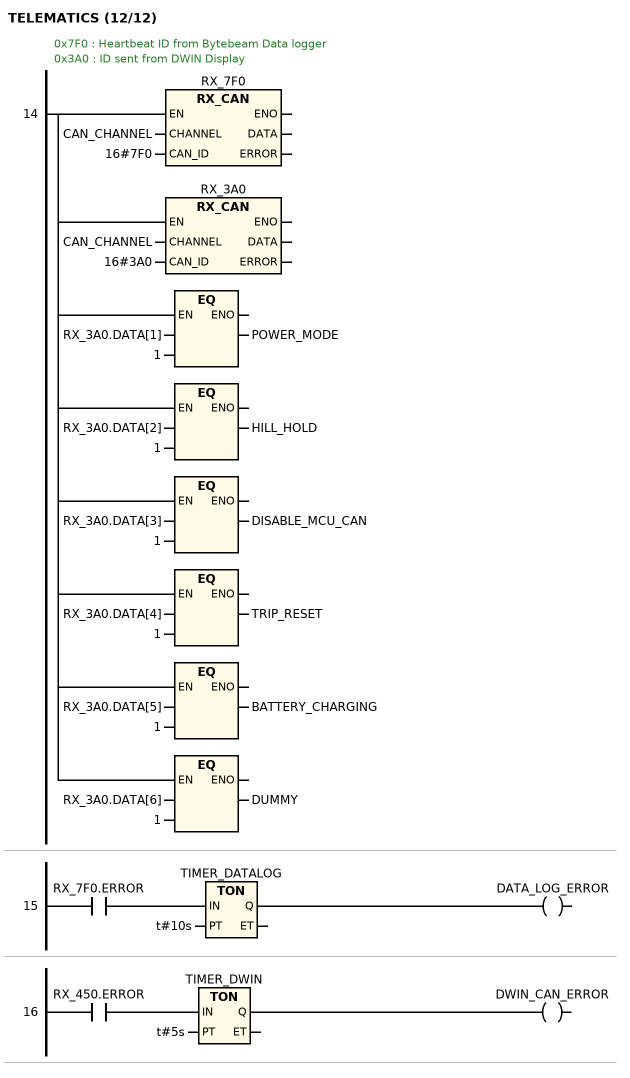
[picture p48: TELEMATICS (LD)]
_LD_ (* Ladder Diagram *)
NETWORK 1 (* CAN ID 301: Battery 1 data Message 1 *)
	*
		EN --- INT_TO_WORD(BATTERY1_POWER) => WB_BATTERY1_POWER.IN_WORD
		EN --- WB_BATTERY1_POWER:WORD_BYTE_CONVERSION(IN_WORD: WB_BATTERY1_POWER.IN_WORD)
		EN --- PACK(BATTERY1_CHARGING, BATTERY1_CAN_ERROR, 0, 0, 0, 0, 0, 0) => PACK_301.B4
		EN --- INT_TO_BYTE(BATTERY1_CAPACITY) => PACK_301.B5
		EN --- PACK_301:PACK_BYTES(B0: BATTERY1_SOC, B1: BATTERY1_SOH, B2: WB_BATTERY1_POWER.BYTE_H, B3: WB_BATTERY1_POWER.BYTE_L, B4: PACK_301.B4, B5: PACK_301.B5, B6: BATTERY1_NTC1, B7: BATTERY1_NTC2) => TX_301.DATA
NETWORK 2 (* CAN ID 303: Battery2 data *)
	*
		EN --- INT_TO_WORD(BATTERY2_POWER) => WB_BATTERY2_POWER.IN_WORD
		EN --- WB_BATTERY2_POWER:WORD_BYTE_CONVERSION(IN_WORD: WB_BATTERY2_POWER.IN_WORD)
		EN --- PACK(BATTERY2_CHARGING, BATTERY2_CAN_ERROR, 0, 0, 0, 0, 0, 0) => PACK_303.B4
		EN --- INT_TO_BYTE(BATTERY2_CAPACITY) => PACK_303.B5
		EN --- PACK_303:PACK_BYTES(B0: BATTERY2_SOC, B1: BATTERY2_SOH, B2: WB_BATTERY2_POWER.BYTE_H, B3: WB_BATTERY2_POWER.BYTE_L, B4: PACK_303.B4, B5: PACK_303.B5, B6: BATTERY2_NTC1, B7: BATTERY2_NTC2) => TX_303.DATA
NETWORK 3 (* CAN ID 305: ODO and TRIP Data *)
	*
		EN --- WB_HYDL_UPTIME:DWORD_BYTE_CONVERSION(INPUT_DWORD: HYDL_UP_TIME)
		EN --- WB_RUNTIME_MIN:DWORD_BYTE_CONVERSION(INPUT_DWORD: RUNTIME)
		EN --- PACK_305:PACK_BYTES(B0: WB_RUNTIME_MIN.BYTE_3, B1: WB_RUNTIME_MIN.BYTE_2, B2: WB_RUNTIME_MIN.BYTE_1, B3: WB_RUNTIME_MIN.BYTE_0, B4: WB_HYDL_UPTIME.BYTE_3, B5: WB_HYDL_UPTIME.BYTE_2, B6: WB_HYDL_UPTIME.BYTE_1, B7: WB_HYDL_UPTIME.BYTE_0) => TX_305.DATA
NETWORK 4 (* CAN ID 306: Basic Vehicle Data *)
	*
		EN --- WB_ODO_METERS:DWORD_BYTE_CONVERSION(INPUT_DWORD: ODO_METER)
		EN --- PACK_306:PACK_BYTES(B0: WB_ODO_METERS.BYTE_3, B1: WB_ODO_METERS.BYTE_2, B2: WB_ODO_METERS.BYTE_1, B3: WB_ODO_METERS.BYTE_0, B4: SPEED, B5: 0, B6: LOG_JX, B7: LOG_JY) => TX_306.DATA
NETWORK 5 (* CAN ID 307: Vehicle Specific parameter frame *)
	*
		EN --- PACK(MCU_IGNITION, NOT KILL_SWITCH, EM_SWITCH, HYDRAULIC_IGNITION, REVERSE, HIGH_SPEED, EM_BRAKE, POWER_MODE) => TX_307.DATA[0]
		EN --- PACK(JOY_ERROR, DATA_LOG_ERROR, DWIN_CAN_ERROR, 0, 0, 0, 0, 0) => TX_307.DATA[1]
		EN --- PACK(BATTERY1_IGNITION, BATTERY2_IGNITION, 0, BATTERY1_RELAY, BATTERY2_RELAY, IMU_ALERT, 0, 0) => TX_307.DATA[2]
		EN --- MOVE(X_ANGLE_BYTE) => TX_307.DATA[6]
		EN --- MOVE(Y_ANGLE_BYTE) => TX_307.DATA[7]
NETWORK 6 (* IMU DATA: 0x308 *)
	*
		EN --- PACK_308:PACK_BYTES(B0: Y_MAX_RETAIN, B1: Y_MIN_RETAIN, B2: X_MAX_RETAIN, B3: X_MIN_RETAIN, B4: Y_MAX_PEAK, B5: Y_MIN_PEAK, B6: X_MAX_PEAK, B7: X_MIN_PEAK) => TX_308.DATA
NETWORK 7 (* 409:- VEHICLE UP TIME (NOT SENDING TO BYTEBEAM) *)
	*
		EN --- WB_VEHICLE_UPTIME:DWORD_BYTE_CONVERSION(INPUT_DWORD: VEHICLE_UP_TIME)
		EN --- WB_VEHICLE_UPTIME_LT:DWORD_BYTE_CONVERSION(INPUT_DWORD: VEHICLE_UP_TIME_LT)
		EN --- PACK_409:PACK_BYTES(B0: WB_VEHICLE_UPTIME_LT.BYTE_3, B1: WB_VEHICLE_UPTIME_LT.BYTE_2, B2: WB_VEHICLE_UPTIME_LT.BYTE_1, B3: WB_VEHICLE_UPTIME_LT.BYTE_0, B4: WB_VEHICLE_UPTIME.BYTE_3, B5: WB_VEHICLE_UPTIME.BYTE_2, B6: WB_VEHICLE_UPTIME.BYTE_1, B7: WB_VEHICLE_UPTIME.BYTE_0) => TX_409.DATA
NETWORK 8 (* CAN ID 310: Motor 41 data Message 1 / CAN ID 311: Motor 41 data Message 2 *)
	*
		EN --- INT_TO_WORD(MOTOR_RPM[1]) => WB_RPM_1.IN_WORD
		EN --- WB_RPM_1:WORD_BYTE_CONVERSION(IN_WORD: WB_RPM_1.IN_WORD, BYTE_L => TX_310.DATA[1]) => TX_310.DATA[0]
		EN --- INT_TO_WORD(MOTOR_POWER[1]) => WB_POWER_1.IN_WORD
		EN --- WB_POWER_1:WORD_BYTE_CONVERSION(IN_WORD: WB_POWER_1.IN_WORD, BYTE_L => TX_310.DATA[3]) => TX_310.DATA[2]
		EN --- WB_PHASE_1:WORD_BYTE_CONVERSION(IN_WORD: MOTOR_PHASE_CURRENT[1], BYTE_L => TX_310.DATA[5]) => TX_310.DATA[4]
		EN --- MOVE(MOTOR_TEMPERATURE[1]) => TX_310.DATA[6]
		EN --- MOVE(MCU_TEMPERATURE[1]) => TX_310.DATA[7]
		EN --- INT_TO_WORD(MOTOR_TARGET_RPM[1]) => WB_TARGET_RPM_1.IN_WORD
		EN --- WB_TARGET_RPM_1:WORD_BYTE_CONVERSION(IN_WORD: WB_TARGET_RPM_1.IN_WORD)
		EN --- WORD_TO_BYTE(MOTOR_OBD_ARRAY[1]) => OBD1_BYTE
		EN --- PACK(MCU_CAN_ERROR[1], 0, 0, 0, 0, 0, 0, 0) => PACK_311.B2
		EN --- PACK_311:PACK_BYTES(B0: WB_TARGET_RPM_1.BYTE_H, B1: WB_TARGET_RPM_1.BYTE_L, B2: PACK_311.B2, B3: OBD1_BYTE, B4: MOTOR1_FAULT_ARRAY[1], B5: MOTOR1_FAULT_ARRAY[2], B6: MOTOR1_FAULT_ARRAY[3], B7: MOTOR1_FAULT_ARRAY[4]) => TX_311.DATA
NETWORK 9 (* CAN ID 312: Motor 42 data Message 1 / CAN ID 313: Motor 42 data Message 2 *)
	*
		EN --- INT_TO_WORD(MOTOR_RPM[2]) => WB_RPM_2.IN_WORD
		EN --- WB_RPM_2:WORD_BYTE_CONVERSION(IN_WORD: WB_RPM_2.IN_WORD, BYTE_L => TX_312.DATA[1]) => TX_312.DATA[0]
		EN --- INT_TO_WORD(MOTOR_POWER[2]) => WB_POWER_2.IN_WORD
		EN --- WB_POWER_2:WORD_BYTE_CONVERSION(IN_WORD: WB_POWER_2.IN_WORD, BYTE_L => TX_312.DATA[3]) => TX_312.DATA[2]
		EN --- WB_PHASE_2:WORD_BYTE_CONVERSION(IN_WORD: MOTOR_PHASE_CURRENT[2], BYTE_L => TX_312.DATA[5]) => TX_312.DATA[4]
		EN --- MOVE(MOTOR_TEMPERATURE[2]) => TX_312.DATA[6]
		EN --- MOVE(MCU_TEMPERATURE[2]) => TX_312.DATA[7]
		EN --- INT_TO_WORD(MOTOR_TARGET_RPM[2]) => WB_TARGET_RPM_2.IN_WORD
		EN --- WB_TARGET_RPM_2:WORD_BYTE_CONVERSION(IN_WORD: WB_TARGET_RPM_2.IN_WORD)
		EN --- WB_OBD_2:WORD_BYTE_CONVERSION(IN_WORD: MOTOR_OBD_ARRAY[2])
		EN --- WORD_TO_BYTE(MOTOR_OBD_ARRAY[2]) => OBD2_BYTE
		EN --- PACK(MCU_CAN_ERROR[2], 0, 0, 0, 0, 0, 0, 0) => TX_313.DATA[2]
		EN --- PACK_313:PACK_BYTES(B0: WB_TARGET_RPM_2.BYTE_H, B1: WB_TARGET_RPM_2.BYTE_L, B2: TX_313.DATA[2], B3: OBD2_BYTE, B4: MOTOR2_FAULT_ARRAY[1], B5: MOTOR2_FAULT_ARRAY[2], B6: MOTOR2_FAULT_ARRAY[3], B7: MOTOR2_FAULT_ARRAY[4]) => TX_313.DATA
NETWORK 10 (* CAN ID 31A: Motor 46 data Message 1 / CAN ID 31B: Motor 46 data Message 2 *)
	*
		EN --- INT_TO_WORD(MOTOR_RPM[6]) => WB_RPM_6.IN_WORD
		EN --- WB_RPM_6:WORD_BYTE_CONVERSION(IN_WORD: WB_RPM_6.IN_WORD, BYTE_L => TX_31A.DATA[1]) => TX_31A.DATA[0]
		EN --- INT_TO_WORD(MOTOR_POWER[6]) => WB_POWER_6.IN_WORD
		EN --- WB_POWER_6:WORD_BYTE_CONVERSION(IN_WORD: WB_POWER_6.IN_WORD, BYTE_L => TX_31A.DATA[3]) => TX_31A.DATA[2]
		EN --- WB_PHASE_6:WORD_BYTE_CONVERSION(IN_WORD: MOTOR_PHASE_CURRENT[6], BYTE_L => TX_31A.DATA[5]) => TX_31A.DATA[4]
		EN --- MOVE(MOTOR_TEMPERATURE[6]) => TX_31A.DATA[6]
		EN --- MOVE(MCU_TEMPERATURE[6]) => TX_31A.DATA[7]
		EN --- INT_TO_WORD(MOTOR_TARGET_RPM[6]) => WB_TARGET_RPM_6.IN_WORD
		EN --- WB_TARGET_RPM_6:WORD_BYTE_CONVERSION(IN_WORD: WB_TARGET_RPM_6.IN_WORD)
		EN --- WB_OBD_6:WORD_BYTE_CONVERSION(IN_WORD: MOTOR_OBD_ARRAY[6])
		EN --- WORD_TO_BYTE(MOTOR_OBD_ARRAY[6]) => OBD6_BYTE
		EN --- PACK(MCU_CAN_ERROR[6], 0, 0, 0, 0, 0, 0, 0) => TX_31B.DATA[2]
		EN --- PACK_31B:PACK_BYTES(B0: WB_TARGET_RPM_6.BYTE_H, B1: WB_TARGET_RPM_6.BYTE_L, B2: TX_31B.DATA[2], B3: OBD6_BYTE, B4: MOTOR6_FAULT_ARRAY[1], B5: MOTOR6_FAULT_ARRAY[2], B6: MOTOR6_FAULT_ARRAY[3], B7: MOTOR6_FAULT_ARRAY[4]) => TX_31B.DATA
NETWORK 11 (* CAN ID 262: BATTERY CHARGING TIME *)
	*
		EN --- REAL_TO_WORD(BATTERY1_FULLCHARGE_MIN) => WD_BATTERY1_FULLCHARGE_MIN
		EN --- REAL_TO_WORD(BATTERY2_FULLCHARGE_MIN) => WD_BATTERY2_FULLCHARGE_MIN
		EN --- WB_FULLCHARGE1_MIN:WORD_BYTE_CONVERSION(IN_WORD: WD_BATTERY1_FULLCHARGE_MIN)
		EN --- WB_FULLCHARGE2_MIN:WORD_BYTE_CONVERSION(IN_WORD: WD_BATTERY2_FULLCHARGE_MIN)
		EN --- PACK_262:PACK_BYTES(B0: WB_FULLCHARGE1_MIN.BYTE_H, B1: WB_FULLCHARGE1_MIN.BYTE_L, B2: WB_FULLCHARGE2_MIN.BYTE_H, B3: WB_FULLCHARGE2_MIN.BYTE_L, B4: 0, B5: 0, B6: 0, B7: 0) => TX_262.DATA
NETWORK 12 (* TO BYTEBEAM *)
	[/TIMER_TX_1.Q] - TIMER_TX_1:TON(IN: *, PT: t#490ms)
		EN --- TX_300:CAN_TX(ENABLE: TRUE, CHANNEL: CAN_CHANNEL, ID: 16#300, DATA: META_FRAME)
		EN --- TX_301:CAN_TX(ENABLE: TRUE, CHANNEL: CAN_CHANNEL, ID: 16#301, DATA: TX_301.DATA)
		EN --- TX_303:CAN_TX(ENABLE: TRUE, CHANNEL: CAN_CHANNEL, ID: 16#303, DATA: TX_303.DATA)
		EN --- TX_306:CAN_TX(ENABLE: TRUE, CHANNEL: CAN_CHANNEL, ID: 16#306, DATA: TX_306.DATA)
		EN --- TX_307:CAN_TX(ENABLE: TRUE, CHANNEL: CAN_CHANNEL, ID: 16#307, DATA: TX_307.DATA)
		EN --- TX_310:CAN_TX(ENABLE: TRUE, CHANNEL: CAN_CHANNEL, ID: 16#310, DATA: TX_310.DATA)
		EN --- TX_311:CAN_TX(ENABLE: TRUE, CHANNEL: CAN_CHANNEL, ID: 16#311, DATA: TX_311.DATA)
		EN --- TX_312:CAN_TX(ENABLE: TRUE, CHANNEL: CAN_CHANNEL, ID: 16#312, DATA: TX_312.DATA)
		EN --- TX_313:CAN_TX(ENABLE: TRUE, CHANNEL: CAN_CHANNEL, ID: 16#313, DATA: TX_313.DATA)
		EN --- TX_31A:CAN_TX(ENABLE: TRUE, CHANNEL: CAN_CHANNEL, ID: 16#31A, DATA: TX_31A.DATA)
		EN --- TX_31B:CAN_TX(ENABLE: TRUE, CHANNEL: CAN_CHANNEL, ID: 16#31B, DATA: TX_31B.DATA)
		EN --- TX_308:CAN_TX(ENABLE: TRUE, CHANNEL: CAN_CHANNEL, ID: 16#308, DATA: TX_308.DATA)
		EN --- TX_305:CAN_TX(ENABLE: TRUE, CHANNEL: CAN_CHANNEL, ID: 16#305, DATA: TX_305.DATA)
NETWORK 13 (* TO DISPLAY *)
	[/TIMER_TX_2.Q] - TIMER_TX_2:TON(IN: *, PT: t#50ms)
		EN --- TX_400:CAN_TX(ENABLE: TRUE, CHANNEL: CAN_CHANNEL, ID: 16#400, DATA: META_FRAME)
		EN --- TX_401:CAN_TX(ENABLE: TRUE, CHANNEL: CAN_CHANNEL, ID: 16#401, DATA: TX_301.DATA)
		EN --- TX_403:CAN_TX(ENABLE: TRUE, CHANNEL: CAN_CHANNEL, ID: 16#403, DATA: TX_303.DATA)
		EN --- TX_406:CAN_TX(ENABLE: TRUE, CHANNEL: CAN_CHANNEL, ID: 16#406, DATA: TX_306.DATA)
		EN --- TX_407:CAN_TX(ENABLE: TRUE, CHANNEL: CAN_CHANNEL, ID: 16#407, DATA: TX_307.DATA)
		EN --- TX_410:CAN_TX(ENABLE: TRUE, CHANNEL: CAN_CHANNEL, ID: 16#410, DATA: TX_310.DATA)
		EN --- TX_411:CAN_TX(ENABLE: TRUE, CHANNEL: CAN_CHANNEL, ID: 16#411, DATA: TX_311.DATA)
		EN --- TX_412:CAN_TX(ENABLE: TRUE, CHANNEL: CAN_CHANNEL, ID: 16#412, DATA: TX_312.DATA)
		EN --- TX_413:CAN_TX(ENABLE: TRUE, CHANNEL: CAN_CHANNEL, ID: 16#413, DATA: TX_313.DATA)
		EN --- TX_41A:CAN_TX(ENABLE: TRUE, CHANNEL: CAN_CHANNEL, ID: 16#41A, DATA: TX_31A.DATA)
		EN --- TX_41B:CAN_TX(ENABLE: TRUE, CHANNEL: CAN_CHANNEL, ID: 16#41B, DATA: TX_31B.DATA)
		EN --- TX_262:CAN_TX(ENABLE: TRUE, CHANNEL: CAN_CHANNEL, ID: 16#262, DATA: TX_262.DATA)
		EN --- TX_408:CAN_TX(ENABLE: TRUE, CHANNEL: CAN_CHANNEL, ID: 16#408, DATA: TX_308.DATA)
		EN --- TX_405:CAN_TX(ENABLE: TRUE, CHANNEL: CAN_CHANNEL, ID: 16#405, DATA: TX_305.DATA)
		EN --- TX_409:CAN_TX(ENABLE: TRUE, CHANNEL: CAN_CHANNEL, ID: 16#409, DATA: TX_409.DATA)
NETWORK 14 (* 0x7F0 : Heartbeat ID from Bytebeam Data logger / 0x3A0 : ID sent from DWIN Display *)
	*
		EN --- RX_7F0:RX_CAN(CHANNEL: CAN_CHANNEL, CAN_ID: 16#7F0)
		EN --- RX_3A0:RX_CAN(CHANNEL: CAN_CHANNEL, CAN_ID: 16#3A0)
		EN --- EQ(RX_3A0.DATA[1], 1) => POWER_MODE
		EN --- EQ(RX_3A0.DATA[2], 1) => HILL_HOLD
		EN --- EQ(RX_3A0.DATA[3], 1) => DISABLE_MCU_CAN
		EN --- EQ(RX_3A0.DATA[4], 1) => TRIP_RESET
		EN --- EQ(RX_3A0.DATA[5], 1) => BATTERY_CHARGING
		EN --- EQ(RX_3A0.DATA[6], 1) => DUMMY
NETWORK 15
	[RX_7F0.ERROR] - TIMER_DATALOG:TON(IN: *, PT: t#10s) --- (DATA_LOG_ERROR)
NETWORK 16
	[RX_450.ERROR] - TIMER_DWIN:TON(IN: *, PT: t#5s) --- (DWIN_CAN_ERROR)
_END_LD_
(* the same logic as Structured Text *)
(* Network 1: CAN ID 301: Battery 1 data Message 1 *)
WB_BATTERY1_POWER.IN_WORD := INT_TO_WORD(BATTERY1_POWER);
WB_BATTERY1_POWER(IN_WORD := WB_BATTERY1_POWER.IN_WORD);
PACK_301.B4 := PACK(BATTERY1_CHARGING, BATTERY1_CAN_ERROR, 0, 0, 0, 0, 0, 0);
PACK_301.B5 := INT_TO_BYTE(BATTERY1_CAPACITY);
PACK_301(B0 := BATTERY1_SOC, B1 := BATTERY1_SOH, B2 := WB_BATTERY1_POWER.BYTE_H, B3 := WB_BATTERY1_POWER.BYTE_L, B4 := PACK_301.B4, B5 := PACK_301.B5, B6 := BATTERY1_NTC1, B7 := BATTERY1_NTC2);
TX_301.DATA := PACK_301.CAN_DATA;
(* Network 2: CAN ID 303: Battery2 data *)
WB_BATTERY2_POWER.IN_WORD := INT_TO_WORD(BATTERY2_POWER);
WB_BATTERY2_POWER(IN_WORD := WB_BATTERY2_POWER.IN_WORD);
PACK_303.B4 := PACK(BATTERY2_CHARGING, BATTERY2_CAN_ERROR, 0, 0, 0, 0, 0, 0);
PACK_303.B5 := INT_TO_BYTE(BATTERY2_CAPACITY);
PACK_303(B0 := BATTERY2_SOC, B1 := BATTERY2_SOH, B2 := WB_BATTERY2_POWER.BYTE_H, B3 := WB_BATTERY2_POWER.BYTE_L, B4 := PACK_303.B4, B5 := PACK_303.B5, B6 := BATTERY2_NTC1, B7 := BATTERY2_NTC2);
TX_303.DATA := PACK_303.CAN_DATA;
(* Network 3: CAN ID 305: ODO and TRIP Data *)
WB_HYDL_UPTIME(INPUT_DWORD := HYDL_UP_TIME);
WB_RUNTIME_MIN(INPUT_DWORD := RUNTIME);
PACK_305(B0 := WB_RUNTIME_MIN.BYTE_3, B1 := WB_RUNTIME_MIN.BYTE_2, B2 := WB_RUNTIME_MIN.BYTE_1, B3 := WB_RUNTIME_MIN.BYTE_0, B4 := WB_HYDL_UPTIME.BYTE_3, B5 := WB_HYDL_UPTIME.BYTE_2, B6 := WB_HYDL_UPTIME.BYTE_1, B7 := WB_HYDL_UPTIME.BYTE_0);
TX_305.DATA := PACK_305.CAN_DATA;
(* Network 4: CAN ID 306: Basic Vehicle Data *)
WB_ODO_METERS(INPUT_DWORD := ODO_METER);
PACK_306(B0 := WB_ODO_METERS.BYTE_3, B1 := WB_ODO_METERS.BYTE_2, B2 := WB_ODO_METERS.BYTE_1, B3 := WB_ODO_METERS.BYTE_0, B4 := SPEED, B5 := 0, B6 := LOG_JX, B7 := LOG_JY);
TX_306.DATA := PACK_306.CAN_DATA;
(* Network 5: CAN ID 307: Vehicle Specific parameter frame *)
TX_307.DATA[0] := PACK(MCU_IGNITION, NOT KILL_SWITCH, EM_SWITCH, HYDRAULIC_IGNITION, REVERSE, HIGH_SPEED, EM_BRAKE, POWER_MODE);
TX_307.DATA[1] := PACK(JOY_ERROR, DATA_LOG_ERROR, DWIN_CAN_ERROR, 0, 0, 0, 0, 0);
TX_307.DATA[2] := PACK(BATTERY1_IGNITION, BATTERY2_IGNITION, 0, BATTERY1_RELAY, BATTERY2_RELAY, IMU_ALERT, 0, 0);
TX_307.DATA[6] := X_ANGLE_BYTE;
TX_307.DATA[7] := Y_ANGLE_BYTE;
(* Network 6: IMU DATA: 0x308 *)
PACK_308(B0 := Y_MAX_RETAIN, B1 := Y_MIN_RETAIN, B2 := X_MAX_RETAIN, B3 := X_MIN_RETAIN, B4 := Y_MAX_PEAK, B5 := Y_MIN_PEAK, B6 := X_MAX_PEAK, B7 := X_MIN_PEAK);
TX_308.DATA := PACK_308.CAN_DATA;
(* Network 7: 409:- VEHICLE UP TIME (NOT SENDING TO BYTEBEAM) *)
WB_VEHICLE_UPTIME(INPUT_DWORD := VEHICLE_UP_TIME);
WB_VEHICLE_UPTIME_LT(INPUT_DWORD := VEHICLE_UP_TIME_LT);
PACK_409(B0 := WB_VEHICLE_UPTIME_LT.BYTE_3, B1 := WB_VEHICLE_UPTIME_LT.BYTE_2, B2 := WB_VEHICLE_UPTIME_LT.BYTE_1, B3 := WB_VEHICLE_UPTIME_LT.BYTE_0, B4 := WB_VEHICLE_UPTIME.BYTE_3, B5 := WB_VEHICLE_UPTIME.BYTE_2, B6 := WB_VEHICLE_UPTIME.BYTE_1, B7 := WB_VEHICLE_UPTIME.BYTE_0);
TX_409.DATA := PACK_409.CAN_DATA;
(* Network 8: CAN ID 310: Motor 41 data Message 1 / CAN ID 311: Motor 41 data Message 2 *)
WB_RPM_1.IN_WORD := INT_TO_WORD(MOTOR_RPM[1]);
WB_RPM_1(IN_WORD := WB_RPM_1.IN_WORD);
TX_310.DATA[1] := WB_RPM_1.BYTE_L;
TX_310.DATA[0] := WB_RPM_1.BYTE_H;
WB_POWER_1.IN_WORD := INT_TO_WORD(MOTOR_POWER[1]);
WB_POWER_1(IN_WORD := WB_POWER_1.IN_WORD);
TX_310.DATA[3] := WB_POWER_1.BYTE_L;
TX_310.DATA[2] := WB_POWER_1.BYTE_H;
WB_PHASE_1(IN_WORD := MOTOR_PHASE_CURRENT[1]);
TX_310.DATA[5] := WB_PHASE_1.BYTE_L;
TX_310.DATA[4] := WB_PHASE_1.BYTE_H;
TX_310.DATA[6] := MOTOR_TEMPERATURE[1];
TX_310.DATA[7] := MCU_TEMPERATURE[1];
WB_TARGET_RPM_1.IN_WORD := INT_TO_WORD(MOTOR_TARGET_RPM[1]);
WB_TARGET_RPM_1(IN_WORD := WB_TARGET_RPM_1.IN_WORD);
OBD1_BYTE := WORD_TO_BYTE(MOTOR_OBD_ARRAY[1]);
PACK_311.B2 := PACK(MCU_CAN_ERROR[1], 0, 0, 0, 0, 0, 0, 0);
PACK_311(B0 := WB_TARGET_RPM_1.BYTE_H, B1 := WB_TARGET_RPM_1.BYTE_L, B2 := PACK_311.B2, B3 := OBD1_BYTE, B4 := MOTOR1_FAULT_ARRAY[1], B5 := MOTOR1_FAULT_ARRAY[2], B6 := MOTOR1_FAULT_ARRAY[3], B7 := MOTOR1_FAULT_ARRAY[4]);
TX_311.DATA := PACK_311.CAN_DATA;
(* Network 9: CAN ID 312: Motor 42 data Message 1 / CAN ID 313: Motor 42 data Message 2 *)
WB_RPM_2.IN_WORD := INT_TO_WORD(MOTOR_RPM[2]);
WB_RPM_2(IN_WORD := WB_RPM_2.IN_WORD);
TX_312.DATA[1] := WB_RPM_2.BYTE_L;
TX_312.DATA[0] := WB_RPM_2.BYTE_H;
WB_POWER_2.IN_WORD := INT_TO_WORD(MOTOR_POWER[2]);
WB_POWER_2(IN_WORD := WB_POWER_2.IN_WORD);
TX_312.DATA[3] := WB_POWER_2.BYTE_L;
TX_312.DATA[2] := WB_POWER_2.BYTE_H;
WB_PHASE_2(IN_WORD := MOTOR_PHASE_CURRENT[2]);
TX_312.DATA[5] := WB_PHASE_2.BYTE_L;
TX_312.DATA[4] := WB_PHASE_2.BYTE_H;
TX_312.DATA[6] := MOTOR_TEMPERATURE[2];
TX_312.DATA[7] := MCU_TEMPERATURE[2];
WB_TARGET_RPM_2.IN_WORD := INT_TO_WORD(MOTOR_TARGET_RPM[2]);
WB_TARGET_RPM_2(IN_WORD := WB_TARGET_RPM_2.IN_WORD);
WB_OBD_2(IN_WORD := MOTOR_OBD_ARRAY[2]);
OBD2_BYTE := WORD_TO_BYTE(MOTOR_OBD_ARRAY[2]);
TX_313.DATA[2] := PACK(MCU_CAN_ERROR[2], 0, 0, 0, 0, 0, 0, 0);
PACK_313(B0 := WB_TARGET_RPM_2.BYTE_H, B1 := WB_TARGET_RPM_2.BYTE_L, B2 := TX_313.DATA[2], B3 := OBD2_BYTE, B4 := MOTOR2_FAULT_ARRAY[1], B5 := MOTOR2_FAULT_ARRAY[2], B6 := MOTOR2_FAULT_ARRAY[3], B7 := MOTOR2_FAULT_ARRAY[4]);
TX_313.DATA := PACK_313.CAN_DATA;
(* Network 10: CAN ID 31A: Motor 46 data Message 1 / CAN ID 31B: Motor 46 data Message 2 *)
WB_RPM_6.IN_WORD := INT_TO_WORD(MOTOR_RPM[6]);
WB_RPM_6(IN_WORD := WB_RPM_6.IN_WORD);
TX_31A.DATA[1] := WB_RPM_6.BYTE_L;
TX_31A.DATA[0] := WB_RPM_6.BYTE_H;
WB_POWER_6.IN_WORD := INT_TO_WORD(MOTOR_POWER[6]);
WB_POWER_6(IN_WORD := WB_POWER_6.IN_WORD);
TX_31A.DATA[3] := WB_POWER_6.BYTE_L;
TX_31A.DATA[2] := WB_POWER_6.BYTE_H;
WB_PHASE_6(IN_WORD := MOTOR_PHASE_CURRENT[6]);
TX_31A.DATA[5] := WB_PHASE_6.BYTE_L;
TX_31A.DATA[4] := WB_PHASE_6.BYTE_H;
TX_31A.DATA[6] := MOTOR_TEMPERATURE[6];
TX_31A.DATA[7] := MCU_TEMPERATURE[6];
WB_TARGET_RPM_6.IN_WORD := INT_TO_WORD(MOTOR_TARGET_RPM[6]);
WB_TARGET_RPM_6(IN_WORD := WB_TARGET_RPM_6.IN_WORD);
WB_OBD_6(IN_WORD := MOTOR_OBD_ARRAY[6]);
OBD6_BYTE := WORD_TO_BYTE(MOTOR_OBD_ARRAY[6]);
TX_31B.DATA[2] := PACK(MCU_CAN_ERROR[6], 0, 0, 0, 0, 0, 0, 0);
PACK_31B(B0 := WB_TARGET_RPM_6.BYTE_H, B1 := WB_TARGET_RPM_6.BYTE_L, B2 := TX_31B.DATA[2], B3 := OBD6_BYTE, B4 := MOTOR6_FAULT_ARRAY[1], B5 := MOTOR6_FAULT_ARRAY[2], B6 := MOTOR6_FAULT_ARRAY[3], B7 := MOTOR6_FAULT_ARRAY[4]);
TX_31B.DATA := PACK_31B.CAN_DATA;
(* Network 11: CAN ID 262: BATTERY CHARGING TIME *)
WD_BATTERY1_FULLCHARGE_MIN := REAL_TO_WORD(BATTERY1_FULLCHARGE_MIN);
WD_BATTERY2_FULLCHARGE_MIN := REAL_TO_WORD(BATTERY2_FULLCHARGE_MIN);
WB_FULLCHARGE1_MIN(IN_WORD := WD_BATTERY1_FULLCHARGE_MIN);
WB_FULLCHARGE2_MIN(IN_WORD := WD_BATTERY2_FULLCHARGE_MIN);
PACK_262(B0 := WB_FULLCHARGE1_MIN.BYTE_H, B1 := WB_FULLCHARGE1_MIN.BYTE_L, B2 := WB_FULLCHARGE2_MIN.BYTE_H, B3 := WB_FULLCHARGE2_MIN.BYTE_L, B4 := 0, B5 := 0, B6 := 0, B7 := 0);
TX_262.DATA := PACK_262.CAN_DATA;
(* Network 12: TO BYTEBEAM *)
TIMER_TX_1(IN := NOT TIMER_TX_1.Q, PT := t#490ms);
IF TIMER_TX_1.Q THEN
	TX_300(ENABLE := TRUE, CHANNEL := CAN_CHANNEL, ID := 16#300, DATA := META_FRAME);
	TX_301(ENABLE := TRUE, CHANNEL := CAN_CHANNEL, ID := 16#301, DATA := TX_301.DATA);
	TX_303(ENABLE := TRUE, CHANNEL := CAN_CHANNEL, ID := 16#303, DATA := TX_303.DATA);
	TX_306(ENABLE := TRUE, CHANNEL := CAN_CHANNEL, ID := 16#306, DATA := TX_306.DATA);
	TX_307(ENABLE := TRUE, CHANNEL := CAN_CHANNEL, ID := 16#307, DATA := TX_307.DATA);
	TX_310(ENABLE := TRUE, CHANNEL := CAN_CHANNEL, ID := 16#310, DATA := TX_310.DATA);
	TX_311(ENABLE := TRUE, CHANNEL := CAN_CHANNEL, ID := 16#311, DATA := TX_311.DATA);
	TX_312(ENABLE := TRUE, CHANNEL := CAN_CHANNEL, ID := 16#312, DATA := TX_312.DATA);
	TX_313(ENABLE := TRUE, CHANNEL := CAN_CHANNEL, ID := 16#313, DATA := TX_313.DATA);
	TX_31A(ENABLE := TRUE, CHANNEL := CAN_CHANNEL, ID := 16#31A, DATA := TX_31A.DATA);
	TX_31B(ENABLE := TRUE, CHANNEL := CAN_CHANNEL, ID := 16#31B, DATA := TX_31B.DATA);
	TX_308(ENABLE := TRUE, CHANNEL := CAN_CHANNEL, ID := 16#308, DATA := TX_308.DATA);
	TX_305(ENABLE := TRUE, CHANNEL := CAN_CHANNEL, ID := 16#305, DATA := TX_305.DATA);
END_IF;
(* Network 13: TO DISPLAY *)
TIMER_TX_2(IN := NOT TIMER_TX_2.Q, PT := t#50ms);
IF TIMER_TX_2.Q THEN
	TX_400(ENABLE := TRUE, CHANNEL := CAN_CHANNEL, ID := 16#400, DATA := META_FRAME);
	TX_401(ENABLE := TRUE, CHANNEL := CAN_CHANNEL, ID := 16#401, DATA := TX_301.DATA);
	TX_403(ENABLE := TRUE, CHANNEL := CAN_CHANNEL, ID := 16#403, DATA := TX_303.DATA);
	TX_406(ENABLE := TRUE, CHANNEL := CAN_CHANNEL, ID := 16#406, DATA := TX_306.DATA);
	TX_407(ENABLE := TRUE, CHANNEL := CAN_CHANNEL, ID := 16#407, DATA := TX_307.DATA);
	TX_410(ENABLE := TRUE, CHANNEL := CAN_CHANNEL, ID := 16#410, DATA := TX_310.DATA);
	TX_411(ENABLE := TRUE, CHANNEL := CAN_CHANNEL, ID := 16#411, DATA := TX_311.DATA);
	TX_412(ENABLE := TRUE, CHANNEL := CAN_CHANNEL, ID := 16#412, DATA := TX_312.DATA);
	TX_413(ENABLE := TRUE, CHANNEL := CAN_CHANNEL, ID := 16#413, DATA := TX_313.DATA);
	TX_41A(ENABLE := TRUE, CHANNEL := CAN_CHANNEL, ID := 16#41A, DATA := TX_31A.DATA);
	TX_41B(ENABLE := TRUE, CHANNEL := CAN_CHANNEL, ID := 16#41B, DATA := TX_31B.DATA);
	TX_262(ENABLE := TRUE, CHANNEL := CAN_CHANNEL, ID := 16#262, DATA := TX_262.DATA);
	TX_408(ENABLE := TRUE, CHANNEL := CAN_CHANNEL, ID := 16#408, DATA := TX_308.DATA);
	TX_405(ENABLE := TRUE, CHANNEL := CAN_CHANNEL, ID := 16#405, DATA := TX_305.DATA);
	TX_409(ENABLE := TRUE, CHANNEL := CAN_CHANNEL, ID := 16#409, DATA := TX_409.DATA);
END_IF;
(* Network 14: 0x7F0 : Heartbeat ID from Bytebeam Data logger / 0x3A0 : ID sent from DWIN Display *)
RX_7F0(CHANNEL := CAN_CHANNEL, CAN_ID := 16#7F0);
RX_3A0(CHANNEL := CAN_CHANNEL, CAN_ID := 16#3A0);
POWER_MODE := RX_3A0.DATA[1] = 1;
HILL_HOLD := RX_3A0.DATA[2] = 1;
DISABLE_MCU_CAN := RX_3A0.DATA[3] = 1;
TRIP_RESET := RX_3A0.DATA[4] = 1;
BATTERY_CHARGING := RX_3A0.DATA[5] = 1;
DUMMY := RX_3A0.DATA[6] = 1;
(* Network 15 *)
TIMER_DATALOG(IN := RX_7F0.ERROR, PT := t#10s);
DATA_LOG_ERROR := TIMER_DATALOG.Q;
(* Network 16 *)
TIMER_DWIN(IN := RX_450.ERROR, PT := t#5s);
DWIN_CAN_ERROR := TIMER_DWIN.Q;
END_PROGRAM

(* POU FB_LIBRARY/DWORD_BYTE_CONVERSION, FBD *)
FUNCTION_BLOCK DWORD_BYTE_CONVERSION
(* BYTE_0 : LSB    ---------   BYTE_3 : MSB *)
VAR_INPUT
	INPUT_DWORD: DWORD;
END_VAR
VAR_OUTPUT
	BYTE_0: BYTE;
	BYTE_1: BYTE;
	BYTE_2: BYTE;
	BYTE_3: BYTE;
END_VAR
VAR
	WORD_1: WORD;
	WORD_2: WORD;
END_VAR
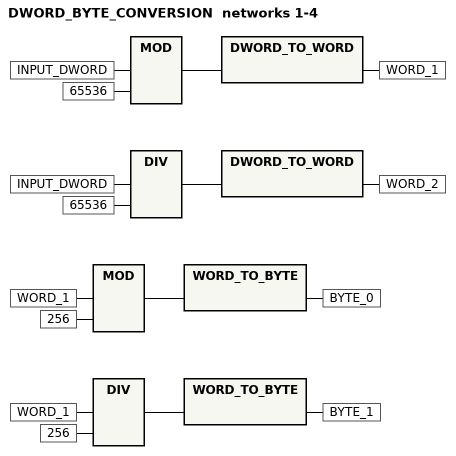
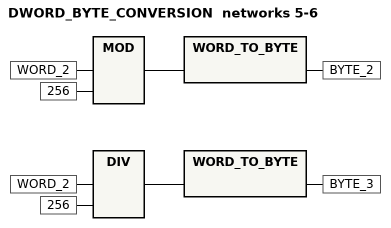
_FBD_ (* Function Block Diagram *)
NETWORK 1
	DWORD_TO_WORD(MOD(INPUT_DWORD, 65536)) => WORD_1
NETWORK 2
	DWORD_TO_WORD(DIV(INPUT_DWORD, 65536)) => WORD_2
NETWORK 3
	WORD_TO_BYTE(MOD(WORD_1, 256)) => BYTE_0
NETWORK 4
	WORD_TO_BYTE(DIV(WORD_1, 256)) => BYTE_1
NETWORK 5
	WORD_TO_BYTE(MOD(WORD_2, 256)) => BYTE_2
NETWORK 6
	WORD_TO_BYTE(DIV(WORD_2, 256)) => BYTE_3
_END_FBD_
(* the same logic as Structured Text *)
(* Network 1 *)
WORD_1 := DWORD_TO_WORD(INPUT_DWORD MOD 65536);
(* Network 2 *)
WORD_2 := DWORD_TO_WORD(INPUT_DWORD / 65536);
(* Network 3 *)
BYTE_0 := WORD_TO_BYTE(WORD_1 MOD 256);
(* Network 4 *)
BYTE_1 := WORD_TO_BYTE(WORD_1 / 256);
(* Network 5 *)
BYTE_2 := WORD_TO_BYTE(WORD_2 MOD 256);
(* Network 6 *)
BYTE_3 := WORD_TO_BYTE(WORD_2 / 256);
END_FUNCTION_BLOCK

(* POU CALCULATIONS, LD *)
PROGRAM CALCULATIONS
VAR
(*SPEED*)
	ABS_RPM1: INT;
	ABS_RPM2: INT;
	RPM_SUM: INT;
	AVG_RPM_REAL: REAL;
	SPEED_REAL: REAL;

(* RUNTIME*)
	MOTOR_1_RUNNING: BOOL;
	MOTOR_2_RUNNING: BOOL;
	HYDRAULIC_HOURS: BOOL;
	COUNT_HOURS: BOOL;
	RISE: R_TRIG;
	FALL: F_TRIG;

	PREVIOUS_TIME: REAL;
	HYDL_PREVIOUS_TIME: REAL;
	VEHICLE_PREVIOUS_TIME: REAL;
	VEHICLE_PREVIOUS_TIME_LT: REAL;

	TON_RUNTIME: TON;
	ET_REAL: REAL;
	HOURS_RUN: REAL;

(*ODO & TRIP*)
	INSTANTANEOUS_DISTANCE: REAL;
	TIMER_ODO: TON;
	ODO_KM_DWORD: DWORD;

(*RANGE*)
	ACTUAL_CAPACITY: REAL;
	ODO_TARGET: DWORD;
	ODO_CYCLE_COMPLETE: BOOL;
	OLD_CAPACITY: REAL;
	DIFFERENCE: REAL;
	CAPACITY_FACTOR: REAL;
	TIMER_RISING: TP;

	HOLD_PREVIOUS_VALUE: BOOL;
	INITIAL_RANGE_REAL: REAL;
	REMAINING_CAPACITY: INT;
	BATTERY1_REMAINING_CAPACITY: INT;
	BATTERY1_FULLCHARGE_HOURS: REAL;
	BATTERY2_REMAINING_CAPACITY: INT;
	BATTERY2_FULLCHARGE_HOURS: REAL;
	TON_HYDL_RUNTIME: TON;
	HYDL_HOURS_RUN: REAL;
	ET_REAL_HYDL: REAL;
	RISE_2: R_TRIG;
	FAL0_2L: F_TRIG;
	FALL_2: F_TRIG;
	ABS_RPM6: INT;
	MINUTE_RUN: REAL;
	ODO_TRIP: DWORD;
	ODO_TRIP_METER: DWORD;
	TRIP_KM_REAL: REAL;
	TRIP_DWORD_KM: DWORD;
	VEHICLE_UP_TIME_COUNT: BOOL;
	RISE_3: R_TRIG;
	FALL_3: F_TRIG;
	TON_VEHICLE_RUNTIME: TON;
	ET_REAL_VEHICLE: REAL;
	VEHICLE_HOURS_RUN: REAL;
	RISE_4: R_TRIG;
	FALL_4: F_TRIG;
	VEHICLE_UP_TIME_COUNT_BW: BOOL;
	VEHICLE_UP_TIME_COUNT_LT: BOOL;
	TON_VEHICLE_RUNTIME_LT: TON;
	ET_REAL_VEHICLE_LT: REAL;
	VEHICLE_HOURS_RUN_LT: REAL;
END_VAR
VAR CONSTANT
	METER_CYCLE: DWORD := 500;						(*CHANGES BASED ON THE CALCULATION OF DISTANCE FACTOR*)
	SPEED_FACTOR: REAL:= 0.00146726;
	ODO_DISTANCE_FACTOR: REAL:= 0.0002037860;	(*GLX with 72.02 Gear Ratio - 500ms Cycle time*)
	ODO_TIME: TIME := T#485MS;							(*Actual calculation factor is for 500ms*)
END_VAR
VAR RETAIN
	RETAIN_DISTANCE: REAL:=457860;							(*In meter*)(*28_03_25 *)
	RETAIN_TIME: REAL := 800640000;			(*222.4 hour- 28-03-25*)	(*Final: REAL:= 3600000 ; //1hour  = 3600000*)
	HYDL_RETAIN_TIME: REAL:=414640000;             (*114.9 HR*)
	VEHICLE_RETAIN_TIME: REAL:=2160000;
	VEHICLE_RETAIN_TIME_LT: REAL:= 801720000;  (*222.7*)
	SUBTRACT_TRIP: DWORD;

END_VAR
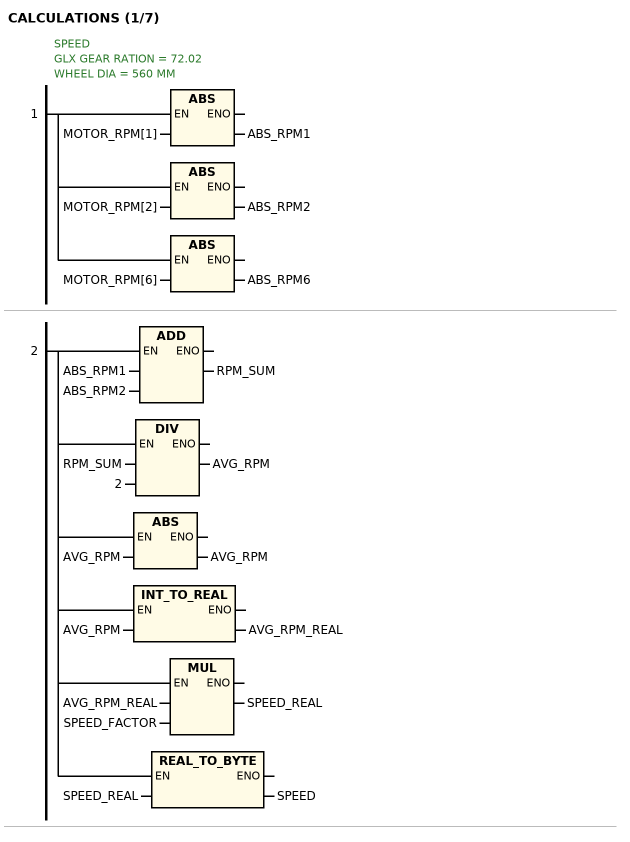
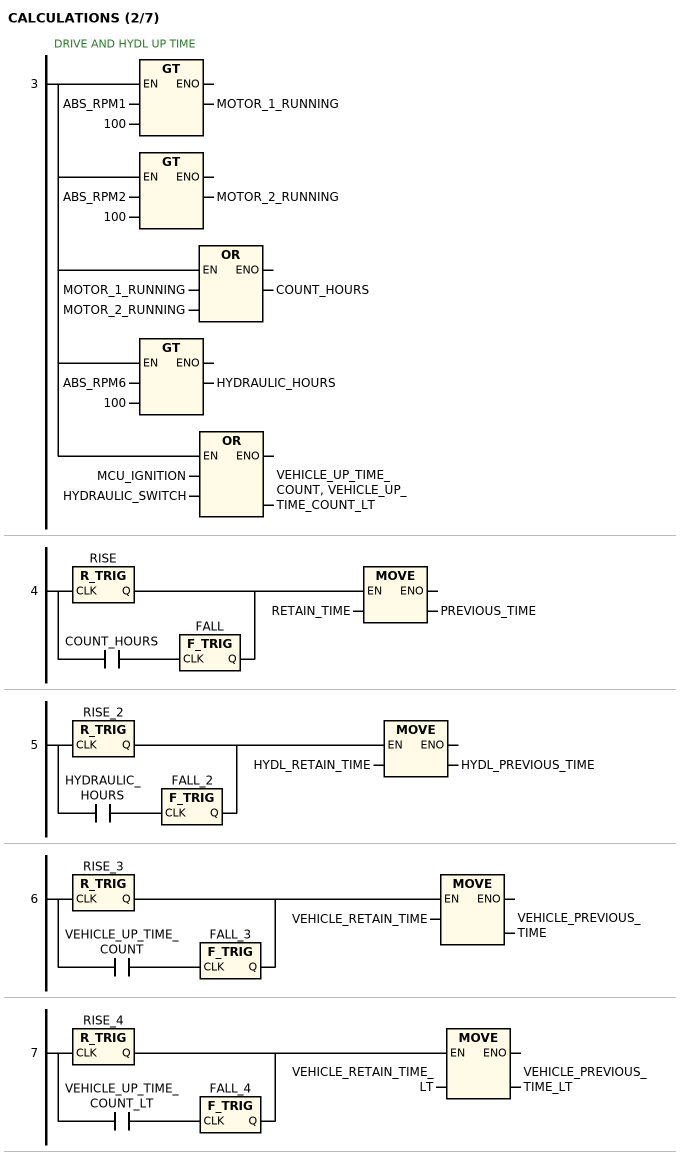
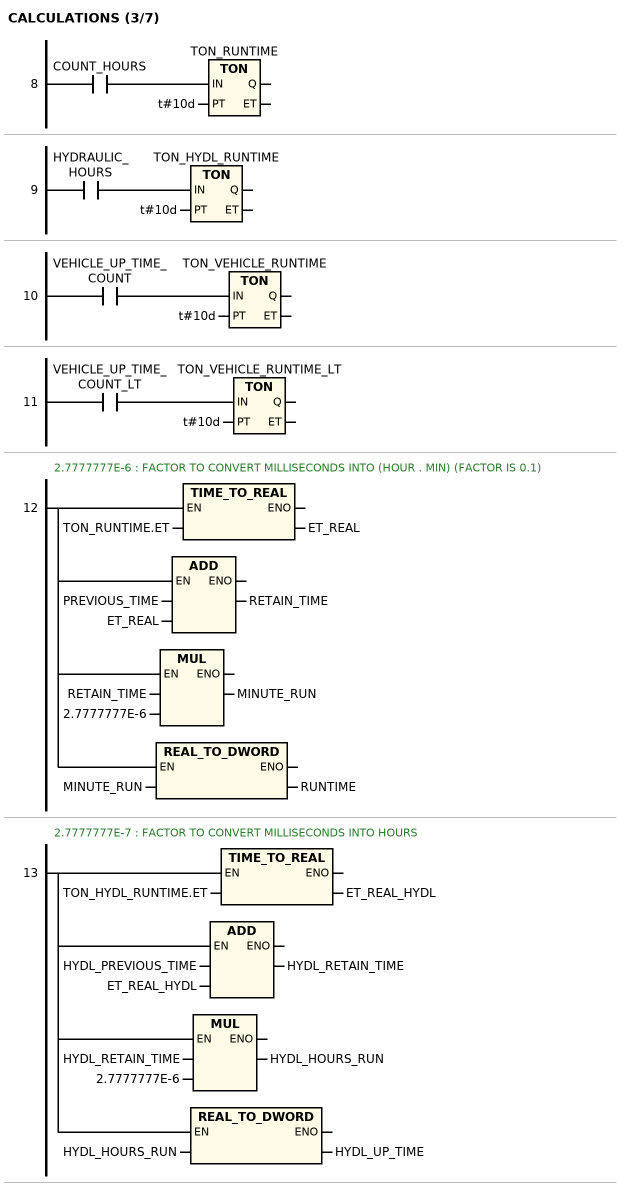
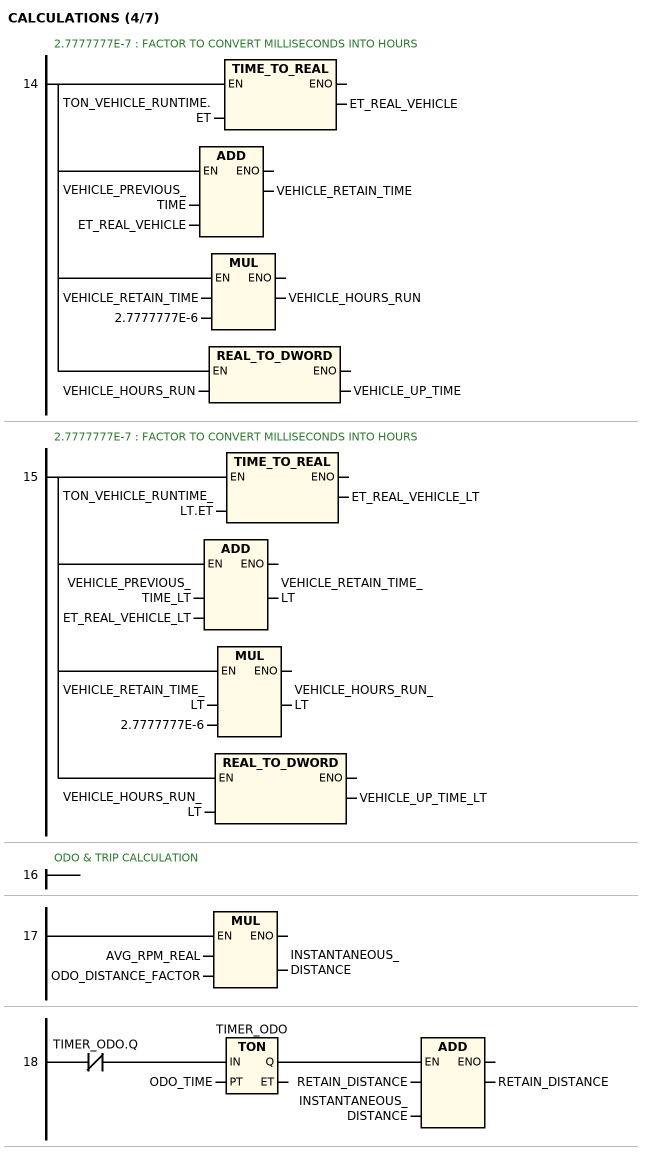
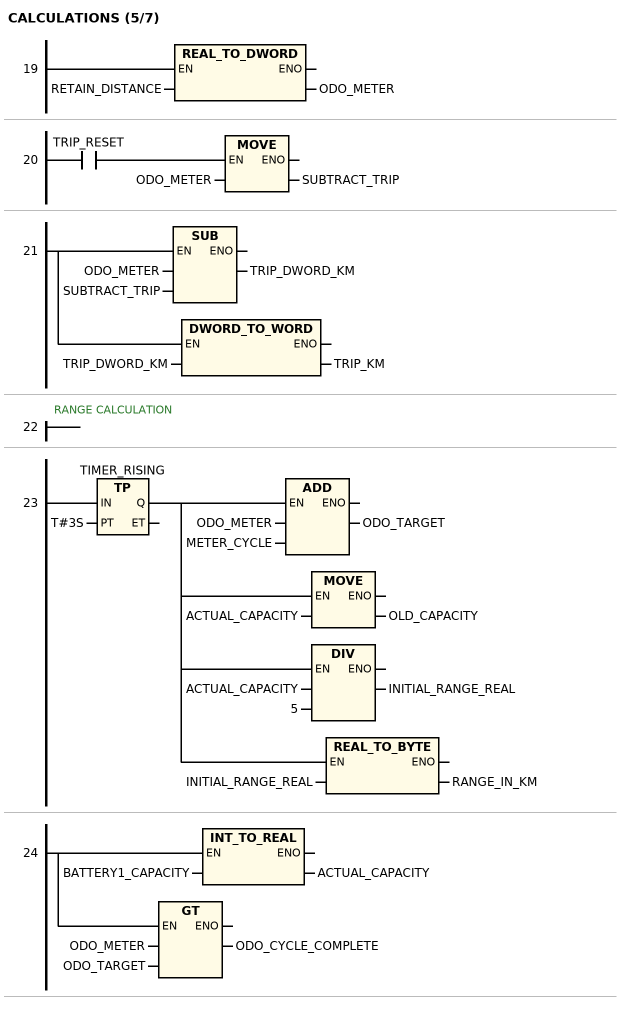
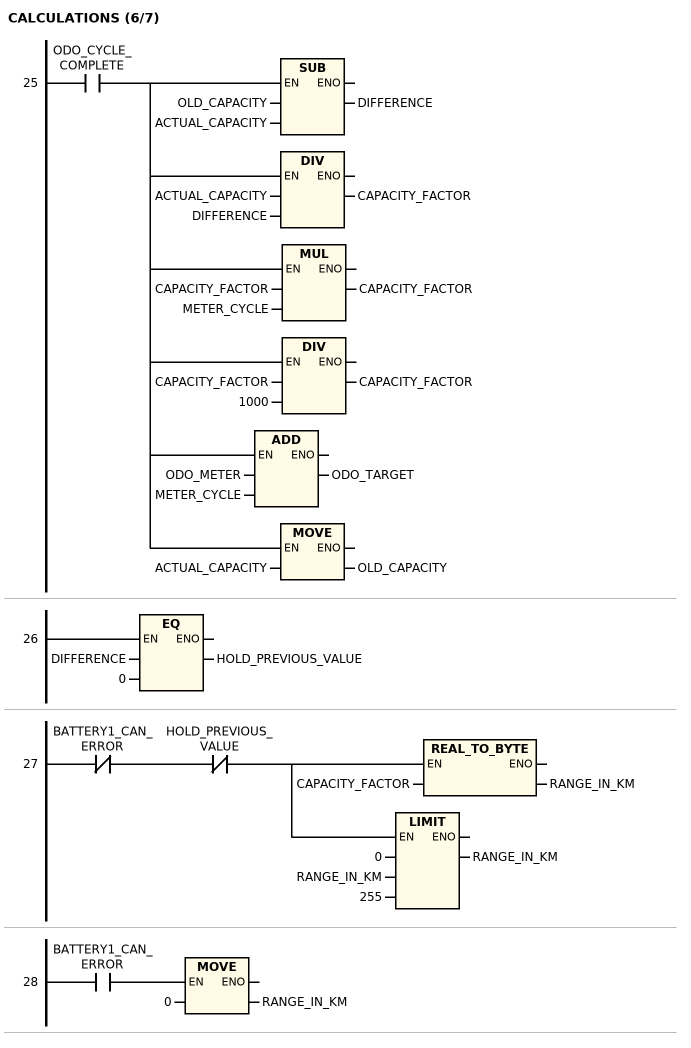
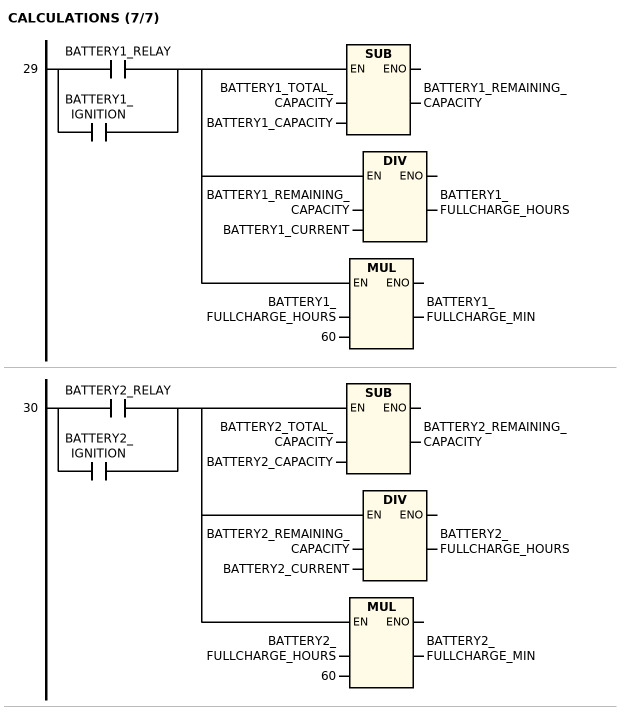
_LD_ (* Ladder Diagram *)
NETWORK 1 (* SPEED / GLX GEAR RATION = 72.02 / WHEEL DIA = 560 MM *)
	*
		EN --- ABS(MOTOR_RPM[1]) => ABS_RPM1
		EN --- ABS(MOTOR_RPM[2]) => ABS_RPM2
		EN --- ABS(MOTOR_RPM[6]) => ABS_RPM6
NETWORK 2
	*
		EN --- ADD(ABS_RPM1, ABS_RPM2) => RPM_SUM
		EN --- DIV(RPM_SUM, 2) => AVG_RPM
		EN --- ABS(AVG_RPM) => AVG_RPM
		EN --- INT_TO_REAL(AVG_RPM) => AVG_RPM_REAL
		EN --- MUL(AVG_RPM_REAL, SPEED_FACTOR) => SPEED_REAL
		EN --- REAL_TO_BYTE(SPEED_REAL) => SPEED
NETWORK 3 (* DRIVE AND HYDL UP TIME *)
	*
		EN --- GT(ABS_RPM1, 100) => MOTOR_1_RUNNING
		EN --- GT(ABS_RPM2, 100) => MOTOR_2_RUNNING
		EN --- OR(MOTOR_1_RUNNING, MOTOR_2_RUNNING) => COUNT_HOURS
		EN --- GT(ABS_RPM6, 100) => HYDRAULIC_HOURS
		EN --- OR(MCU_IGNITION, HYDRAULIC_SWITCH) => VEHICLE_UP_TIME_COUNT, VEHICLE_UP_TIME_COUNT_LT
NETWORK 4
	{ RISE:R_TRIG(CLK: *) | [COUNT_HOURS] - FALL:F_TRIG(CLK: *) }
		EN --- MOVE(RETAIN_TIME) => PREVIOUS_TIME
NETWORK 5
	{ RISE_2:R_TRIG(CLK: *) | [HYDRAULIC_HOURS] - FALL_2:F_TRIG(CLK: *) }
		EN --- MOVE(HYDL_RETAIN_TIME) => HYDL_PREVIOUS_TIME
NETWORK 6
	{ RISE_3:R_TRIG(CLK: *) | [VEHICLE_UP_TIME_COUNT] - FALL_3:F_TRIG(CLK: *) }
		EN --- MOVE(VEHICLE_RETAIN_TIME) => VEHICLE_PREVIOUS_TIME
NETWORK 7
	{ RISE_4:R_TRIG(CLK: *) | [VEHICLE_UP_TIME_COUNT_LT] - FALL_4:F_TRIG(CLK: *) }
		EN --- MOVE(VEHICLE_RETAIN_TIME_LT) => VEHICLE_PREVIOUS_TIME_LT
NETWORK 8
	[COUNT_HOURS] - TON_RUNTIME:TON(IN: *, PT: t#10d)
NETWORK 9
	[HYDRAULIC_HOURS] - TON_HYDL_RUNTIME:TON(IN: *, PT: t#10d)
NETWORK 10
	[VEHICLE_UP_TIME_COUNT] - TON_VEHICLE_RUNTIME:TON(IN: *, PT: t#10d)
NETWORK 11
	[VEHICLE_UP_TIME_COUNT_LT] - TON_VEHICLE_RUNTIME_LT:TON(IN: *, PT: t#10d)
NETWORK 12 (* 2.7777777E-6 : FACTOR TO CONVERT MILLISECONDS INTO (HOUR . MIN) (FACTOR IS 0.1) *)
	*
		EN --- TIME_TO_REAL(TON_RUNTIME.ET) => ET_REAL
		EN --- ADD(PREVIOUS_TIME, ET_REAL) => RETAIN_TIME
		EN --- MUL(RETAIN_TIME, 2.7777777E-6) => MINUTE_RUN
		EN --- REAL_TO_DWORD(MINUTE_RUN) => RUNTIME
NETWORK 13 (* 2.7777777E-7 : FACTOR TO CONVERT MILLISECONDS INTO HOURS *)
	*
		EN --- TIME_TO_REAL(TON_HYDL_RUNTIME.ET) => ET_REAL_HYDL
		EN --- ADD(HYDL_PREVIOUS_TIME, ET_REAL_HYDL) => HYDL_RETAIN_TIME
		EN --- MUL(HYDL_RETAIN_TIME, 2.7777777E-6) => HYDL_HOURS_RUN
		EN --- REAL_TO_DWORD(HYDL_HOURS_RUN) => HYDL_UP_TIME
NETWORK 14 (* 2.7777777E-7 : FACTOR TO CONVERT MILLISECONDS INTO HOURS *)
	*
		EN --- TIME_TO_REAL(TON_VEHICLE_RUNTIME.ET) => ET_REAL_VEHICLE
		EN --- ADD(VEHICLE_PREVIOUS_TIME, ET_REAL_VEHICLE) => VEHICLE_RETAIN_TIME
		EN --- MUL(VEHICLE_RETAIN_TIME, 2.7777777E-6) => VEHICLE_HOURS_RUN
		EN --- REAL_TO_DWORD(VEHICLE_HOURS_RUN) => VEHICLE_UP_TIME
NETWORK 15 (* 2.7777777E-7 : FACTOR TO CONVERT MILLISECONDS INTO HOURS *)
	*
		EN --- TIME_TO_REAL(TON_VEHICLE_RUNTIME_LT.ET) => ET_REAL_VEHICLE_LT
		EN --- ADD(VEHICLE_PREVIOUS_TIME_LT, ET_REAL_VEHICLE_LT) => VEHICLE_RETAIN_TIME_LT
		EN --- MUL(VEHICLE_RETAIN_TIME_LT, 2.7777777E-6) => VEHICLE_HOURS_RUN_LT
		EN --- REAL_TO_DWORD(VEHICLE_HOURS_RUN_LT) => VEHICLE_UP_TIME_LT
NETWORK 16 (* ODO & TRIP CALCULATION *)
	*
NETWORK 17
	*
		EN --- MUL(AVG_RPM_REAL, ODO_DISTANCE_FACTOR) => INSTANTANEOUS_DISTANCE
NETWORK 18
	[/TIMER_ODO.Q] - TIMER_ODO:TON(IN: *, PT: ODO_TIME)
		EN --- ADD(RETAIN_DISTANCE, INSTANTANEOUS_DISTANCE) => RETAIN_DISTANCE
NETWORK 19
	*
		EN --- REAL_TO_DWORD(RETAIN_DISTANCE) => ODO_METER
NETWORK 20
	[TRIP_RESET]
		EN --- MOVE(ODO_METER) => SUBTRACT_TRIP
NETWORK 21
	*
		EN --- SUB(ODO_METER, SUBTRACT_TRIP) => TRIP_DWORD_KM
		EN --- DWORD_TO_WORD(TRIP_DWORD_KM) => TRIP_KM
NETWORK 22 (* RANGE CALCULATION *)
	*
NETWORK 23
	TIMER_RISING:TP(IN: *, PT: T#3S)
		EN --- ADD(ODO_METER, METER_CYCLE) => ODO_TARGET
		EN --- MOVE(ACTUAL_CAPACITY) => OLD_CAPACITY
		EN --- DIV(ACTUAL_CAPACITY, 5) => INITIAL_RANGE_REAL
		EN --- REAL_TO_BYTE(INITIAL_RANGE_REAL) => RANGE_IN_KM
NETWORK 24
	*
		EN --- INT_TO_REAL(BATTERY1_CAPACITY) => ACTUAL_CAPACITY
		EN --- GT(ODO_METER, ODO_TARGET) => ODO_CYCLE_COMPLETE
NETWORK 25
	[ODO_CYCLE_COMPLETE]
		EN --- SUB(OLD_CAPACITY, ACTUAL_CAPACITY) => DIFFERENCE
		EN --- DIV(ACTUAL_CAPACITY, DIFFERENCE) => CAPACITY_FACTOR
		EN --- MUL(CAPACITY_FACTOR, METER_CYCLE) => CAPACITY_FACTOR
		EN --- DIV(CAPACITY_FACTOR, 1000) => CAPACITY_FACTOR
		EN --- ADD(ODO_METER, METER_CYCLE) => ODO_TARGET
		EN --- MOVE(ACTUAL_CAPACITY) => OLD_CAPACITY
NETWORK 26
	*
		EN --- EQ(DIFFERENCE, 0) => HOLD_PREVIOUS_VALUE
NETWORK 27
	[/BATTERY1_CAN_ERROR] - [/HOLD_PREVIOUS_VALUE]
		EN --- REAL_TO_BYTE(CAPACITY_FACTOR) => RANGE_IN_KM
		EN --- LIMIT(0, RANGE_IN_KM, 255) => RANGE_IN_KM
NETWORK 28
	[BATTERY1_CAN_ERROR]
		EN --- MOVE(0) => RANGE_IN_KM
NETWORK 29
	{ [BATTERY1_RELAY] | [BATTERY1_IGNITION] }
		EN --- SUB(BATTERY1_TOTAL_CAPACITY, BATTERY1_CAPACITY) => BATTERY1_REMAINING_CAPACITY
		EN --- DIV(BATTERY1_REMAINING_CAPACITY, BATTERY1_CURRENT) => BATTERY1_FULLCHARGE_HOURS
		EN --- MUL(BATTERY1_FULLCHARGE_HOURS, 60) => BATTERY1_FULLCHARGE_MIN
NETWORK 30
	{ [BATTERY2_RELAY] | [BATTERY2_IGNITION] }
		EN --- SUB(BATTERY2_TOTAL_CAPACITY, BATTERY2_CAPACITY) => BATTERY2_REMAINING_CAPACITY
		EN --- DIV(BATTERY2_REMAINING_CAPACITY, BATTERY2_CURRENT) => BATTERY2_FULLCHARGE_HOURS
		EN --- MUL(BATTERY2_FULLCHARGE_HOURS, 60) => BATTERY2_FULLCHARGE_MIN
_END_LD_
(* the same logic as Structured Text *)
(* Network 1 *)
ABS_RPM1 := ABS(MOTOR_RPM[1]);
ABS_RPM2 := ABS(MOTOR_RPM[2]);
ABS_RPM6 := ABS(MOTOR_RPM[6]);
(* Network 2 *)
RPM_SUM := ABS_RPM1 + ABS_RPM2;
AVG_RPM := RPM_SUM / 2;
AVG_RPM := ABS(AVG_RPM);
AVG_RPM_REAL := INT_TO_REAL(AVG_RPM);
SPEED_REAL := AVG_RPM_REAL * SPEED_FACTOR;
SPEED := REAL_TO_BYTE(SPEED_REAL);
(* Network 3: see the listing above *)
(* Network 4 *)
RISE(CLK := TRUE);
FALL(CLK := COUNT_HOURS);
IF RISE.Q OR FALL.Q THEN
	PREVIOUS_TIME := RETAIN_TIME;
END_IF;
(* Network 5 *)
RISE_2(CLK := TRUE);
FALL_2(CLK := HYDRAULIC_HOURS);
IF RISE_2.Q OR FALL_2.Q THEN
	HYDL_PREVIOUS_TIME := HYDL_RETAIN_TIME;
END_IF;
(* Network 6 *)
RISE_3(CLK := TRUE);
FALL_3(CLK := VEHICLE_UP_TIME_COUNT);
IF RISE_3.Q OR FALL_3.Q THEN
	VEHICLE_PREVIOUS_TIME := VEHICLE_RETAIN_TIME;
END_IF;
(* Network 7 *)
RISE_4(CLK := TRUE);
FALL_4(CLK := VEHICLE_UP_TIME_COUNT_LT);
IF RISE_4.Q OR FALL_4.Q THEN
	VEHICLE_PREVIOUS_TIME_LT := VEHICLE_RETAIN_TIME_LT;
END_IF;
(* Network 8 *)
TON_RUNTIME(IN := COUNT_HOURS, PT := t#10d);
(* Network 9 *)
TON_HYDL_RUNTIME(IN := HYDRAULIC_HOURS, PT := t#10d);
(* Network 10 *)
TON_VEHICLE_RUNTIME(IN := VEHICLE_UP_TIME_COUNT, PT := t#10d);
(* Network 11 *)
TON_VEHICLE_RUNTIME_LT(IN := VEHICLE_UP_TIME_COUNT_LT, PT := t#10d);
(* Network 12 *)
ET_REAL := TIME_TO_REAL(TON_RUNTIME.ET);
RETAIN_TIME := PREVIOUS_TIME + ET_REAL;
MINUTE_RUN := RETAIN_TIME * (2.7777777E-6);
RUNTIME := REAL_TO_DWORD(MINUTE_RUN);
(* Network 13 *)
ET_REAL_HYDL := TIME_TO_REAL(TON_HYDL_RUNTIME.ET);
HYDL_RETAIN_TIME := HYDL_PREVIOUS_TIME + ET_REAL_HYDL;
HYDL_HOURS_RUN := HYDL_RETAIN_TIME * (2.7777777E-6);
HYDL_UP_TIME := REAL_TO_DWORD(HYDL_HOURS_RUN);
(* Network 14 *)
ET_REAL_VEHICLE := TIME_TO_REAL(TON_VEHICLE_RUNTIME.ET);
VEHICLE_RETAIN_TIME := VEHICLE_PREVIOUS_TIME + ET_REAL_VEHICLE;
VEHICLE_HOURS_RUN := VEHICLE_RETAIN_TIME * (2.7777777E-6);
VEHICLE_UP_TIME := REAL_TO_DWORD(VEHICLE_HOURS_RUN);
(* Network 15 *)
ET_REAL_VEHICLE_LT := TIME_TO_REAL(TON_VEHICLE_RUNTIME_LT.ET);
VEHICLE_RETAIN_TIME_LT := VEHICLE_PREVIOUS_TIME_LT + ET_REAL_VEHICLE_LT;
VEHICLE_HOURS_RUN_LT := VEHICLE_RETAIN_TIME_LT * (2.7777777E-6);
VEHICLE_UP_TIME_LT := REAL_TO_DWORD(VEHICLE_HOURS_RUN_LT);
(* Network 16: see the listing above *)
(* Network 17 *)
INSTANTANEOUS_DISTANCE := AVG_RPM_REAL * ODO_DISTANCE_FACTOR;
(* Network 18 *)
TIMER_ODO(IN := NOT TIMER_ODO.Q, PT := ODO_TIME);
IF TIMER_ODO.Q THEN
	RETAIN_DISTANCE := RETAIN_DISTANCE + INSTANTANEOUS_DISTANCE;
END_IF;
(* Network 19 *)
ODO_METER := REAL_TO_DWORD(RETAIN_DISTANCE);
(* Network 20 *)
IF TRIP_RESET THEN
	SUBTRACT_TRIP := ODO_METER;
END_IF;
(* Network 21 *)
TRIP_DWORD_KM := ODO_METER - SUBTRACT_TRIP;
TRIP_KM := DWORD_TO_WORD(TRIP_DWORD_KM);
(* Network 22: see the listing above *)
(* Network 23 *)
TIMER_RISING(IN := TRUE, PT := T#3S);
IF TIMER_RISING.Q THEN
	ODO_TARGET := ODO_METER + METER_CYCLE;
	OLD_CAPACITY := ACTUAL_CAPACITY;
	INITIAL_RANGE_REAL := ACTUAL_CAPACITY / 5;
	RANGE_IN_KM := REAL_TO_BYTE(INITIAL_RANGE_REAL);
END_IF;
(* Network 24 *)
ACTUAL_CAPACITY := INT_TO_REAL(BATTERY1_CAPACITY);
ODO_CYCLE_COMPLETE := ODO_METER > ODO_TARGET;
(* Network 25 *)
IF ODO_CYCLE_COMPLETE THEN
	DIFFERENCE := OLD_CAPACITY - ACTUAL_CAPACITY;
	CAPACITY_FACTOR := ACTUAL_CAPACITY / DIFFERENCE;
	CAPACITY_FACTOR := CAPACITY_FACTOR * METER_CYCLE;
	CAPACITY_FACTOR := CAPACITY_FACTOR / 1000;
	ODO_TARGET := ODO_METER + METER_CYCLE;
	OLD_CAPACITY := ACTUAL_CAPACITY;
END_IF;
(* Network 26 *)
HOLD_PREVIOUS_VALUE := DIFFERENCE = 0;
(* Network 27 *)
IF NOT BATTERY1_CAN_ERROR AND NOT HOLD_PREVIOUS_VALUE THEN
	RANGE_IN_KM := REAL_TO_BYTE(CAPACITY_FACTOR);
	RANGE_IN_KM := LIMIT(0, RANGE_IN_KM, 255);
END_IF;
(* Network 28 *)
IF BATTERY1_CAN_ERROR THEN
	RANGE_IN_KM := 0;
END_IF;
(* Network 29 *)
IF BATTERY1_RELAY OR BATTERY1_IGNITION THEN
	BATTERY1_REMAINING_CAPACITY := BATTERY1_TOTAL_CAPACITY - BATTERY1_CAPACITY;
	BATTERY1_FULLCHARGE_HOURS := BATTERY1_REMAINING_CAPACITY / BATTERY1_CURRENT;
	BATTERY1_FULLCHARGE_MIN := BATTERY1_FULLCHARGE_HOURS * 60;
END_IF;
(* Network 30 *)
IF BATTERY2_RELAY OR BATTERY2_IGNITION THEN
	BATTERY2_REMAINING_CAPACITY := BATTERY2_TOTAL_CAPACITY - BATTERY2_CAPACITY;
	BATTERY2_FULLCHARGE_HOURS := BATTERY2_REMAINING_CAPACITY / BATTERY2_CURRENT;
	BATTERY2_FULLCHARGE_MIN := BATTERY2_FULLCHARGE_HOURS * 60;
END_IF;
END_PROGRAM

(* POU PROGRAM_FBs/CLN_BATTERY_SELECTION_2, LD *)
 FUNCTION_BLOCK CLN_BATTERY_SELECTION_2
VAR_INPUT
	BAT_SOC: BYTE;
	BAT_SOH: BYTE;
	BAT_POWER: INT;
	BAT_NTC1: BYTE;
	BAT_NTC2: BYTE;
	BAT_CAN_ERROR: BOOL;
	BAT_CURRENT: INT;
END_VAR
VAR_OUTPUT
END_VAR
VAR
	BAT1_TON: TON;
	BAT2_TON: TON;
END_VAR
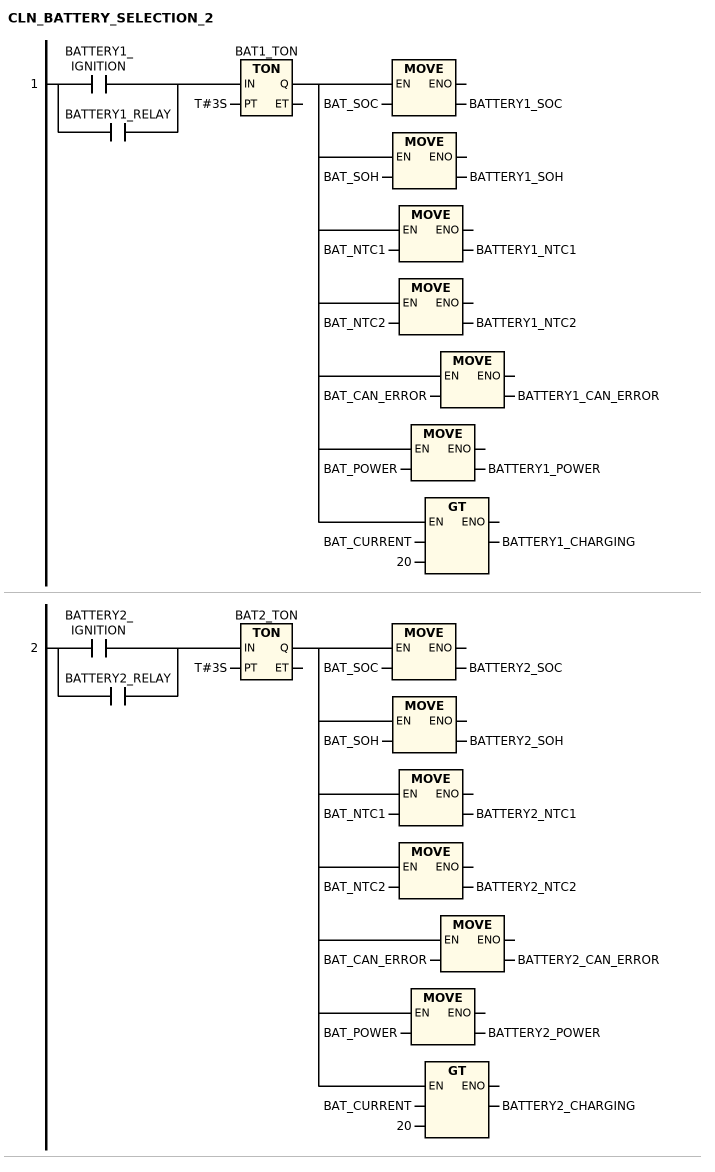
_LD_ (* Ladder Diagram *)
NETWORK 1
	{ [BATTERY1_IGNITION] | [BATTERY1_RELAY] } - BAT1_TON:TON(IN: *, PT: T#3S)
		EN --- MOVE(BAT_SOC) => BATTERY1_SOC
		EN --- MOVE(BAT_SOH) => BATTERY1_SOH
		EN --- MOVE(BAT_NTC1) => BATTERY1_NTC1
		EN --- MOVE(BAT_NTC2) => BATTERY1_NTC2
		EN --- MOVE(BAT_CAN_ERROR) => BATTERY1_CAN_ERROR
		EN --- MOVE(BAT_POWER) => BATTERY1_POWER
		EN --- GT(BAT_CURRENT, 20) => BATTERY1_CHARGING
NETWORK 2
	{ [BATTERY2_IGNITION] | [BATTERY2_RELAY] } - BAT2_TON:TON(IN: *, PT: T#3S)
		EN --- MOVE(BAT_SOC) => BATTERY2_SOC
		EN --- MOVE(BAT_SOH) => BATTERY2_SOH
		EN --- MOVE(BAT_NTC1) => BATTERY2_NTC1
		EN --- MOVE(BAT_NTC2) => BATTERY2_NTC2
		EN --- MOVE(BAT_CAN_ERROR) => BATTERY2_CAN_ERROR
		EN --- MOVE(BAT_POWER) => BATTERY2_POWER
		EN --- GT(BAT_CURRENT, 20) => BATTERY2_CHARGING
_END_LD_
(* the same logic as Structured Text *)
(* Network 1 *)
BAT1_TON(IN := BATTERY1_IGNITION OR BATTERY1_RELAY, PT := T#3S);
IF BAT1_TON.Q THEN
	BATTERY1_SOC := BAT_SOC;
	BATTERY1_SOH := BAT_SOH;
	BATTERY1_NTC1 := BAT_NTC1;
	BATTERY1_NTC2 := BAT_NTC2;
	BATTERY1_CAN_ERROR := BAT_CAN_ERROR;
	BATTERY1_POWER := BAT_POWER;
	BATTERY1_CHARGING := BAT_CURRENT > 20;
END_IF;
(* Network 2 *)
BAT2_TON(IN := BATTERY2_IGNITION OR BATTERY2_RELAY, PT := T#3S);
IF BAT2_TON.Q THEN
	BATTERY2_SOC := BAT_SOC;
	BATTERY2_SOH := BAT_SOH;
	BATTERY2_NTC1 := BAT_NTC1;
	BATTERY2_NTC2 := BAT_NTC2;
	BATTERY2_CAN_ERROR := BAT_CAN_ERROR;
	BATTERY2_POWER := BAT_POWER;
	BATTERY2_CHARGING := BAT_CURRENT > 20;
END_IF;
END_FUNCTION_BLOCK

(* POU PROGRAM_FBs/CLN_BATTERY_SWITCH, LD *)
FUNCTION_BLOCK CLN_BATTERY_SWITCH

(*THIS BLOCK IS COMPATIBLE FOR 2X CLN BATTERIES*)

VAR_INPUT
	CHARGER_IN: BOOL;
	IGN_KEY: BOOL;
	BAT1_IGNITION: BOOL;
	BAT2_IGNITION: BOOL;
	SOC_BAT1: BYTE;
	SOC_BAT2: BYTE;
	BAT1_CAN_ERROR: BOOL;
	BAT2_CAN_ERROR: BOOL;
END_VAR

VAR_OUTPUT
	RELAY_BAT1: BOOL;
	RELAY_BAT2: BOOL;
	ERROR: BOOL;
END_VAR

VAR
	BAT1_CAN_TIMER: TON;
	BAT2_CAN_TIMER: TON;
	BAT1_FULL: BOOL;
	BAT2_FULL: BOOL;
	BAT1_80: BOOL;
	BAT2_80: BOOL;
	CHARGE_1: BOOL;
	RELAY1_TIMER: TON;
	RELAY2_TIMER: TON;
	BLUE_BLINK: BLINK;
	CHARGE1_BLINK: BLINK;
	CHARGE2_BLINK: BLINK;
	CHARGING_SAFETY: BOOL;

	ERROR_TIMER: TON;
END_VAR
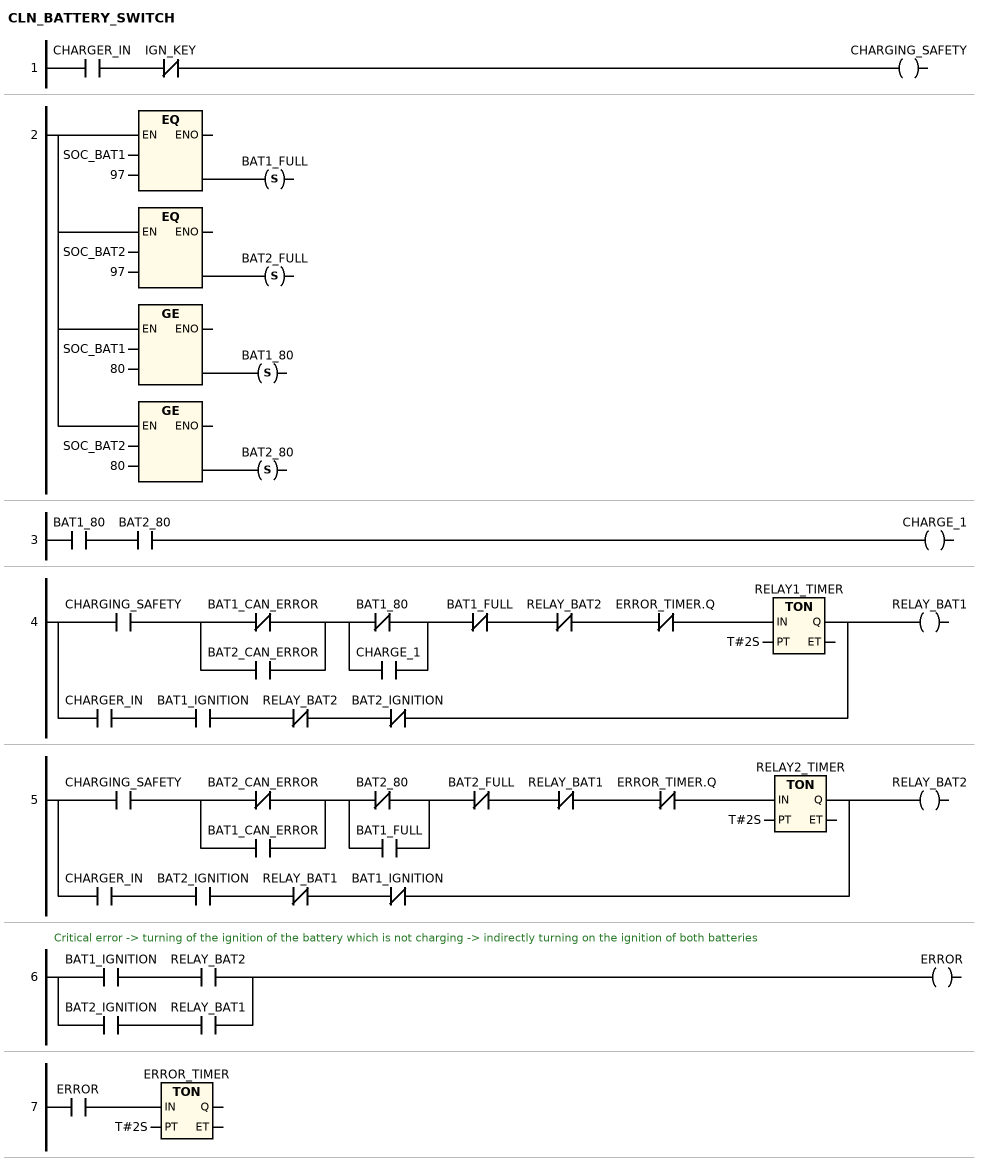
_LD_ (* Ladder Diagram *)
NETWORK 1
	[CHARGER_IN] - [/IGN_KEY] --- (CHARGING_SAFETY)
NETWORK 2
	*
		EN --- EQ(SOC_BAT1, 97) => S BAT1_FULL
		EN --- EQ(SOC_BAT2, 97) => S BAT2_FULL
		EN --- GE(SOC_BAT1, 80) => S BAT1_80
		EN --- GE(SOC_BAT2, 80) => S BAT2_80
NETWORK 3
	[BAT1_80] - [BAT2_80] --- (CHARGE_1)
NETWORK 4
	{ [CHARGING_SAFETY] - { [/BAT1_CAN_ERROR] | [BAT2_CAN_ERROR] } - { [/BAT1_80] | [CHARGE_1] } - [/BAT1_FULL] - [/RELAY_BAT2] - [/ERROR_TIMER.Q] - RELAY1_TIMER:TON(IN: *, PT: T#2S) | [CHARGER_IN] - [BAT1_IGNITION] - [/RELAY_BAT2] - [/BAT2_IGNITION] } --- (RELAY_BAT1)
NETWORK 5
	{ [CHARGING_SAFETY] - { [/BAT2_CAN_ERROR] | [BAT1_CAN_ERROR] } - { [/BAT2_80] | [BAT1_FULL] } - [/BAT2_FULL] - [/RELAY_BAT1] - [/ERROR_TIMER.Q] - RELAY2_TIMER:TON(IN: *, PT: T#2S) | [CHARGER_IN] - [BAT2_IGNITION] - [/RELAY_BAT1] - [/BAT1_IGNITION] } --- (RELAY_BAT2)
NETWORK 6 (* Critical error -> turning of the ignition of the battery which is not charging -> indirectly turning on the ignition of both batteries *)
	{ [BAT1_IGNITION] - [RELAY_BAT2] | [BAT2_IGNITION] - [RELAY_BAT1] } --- (ERROR)
NETWORK 7
	[ERROR] - ERROR_TIMER:TON(IN: *, PT: T#2S)
_END_LD_
(* the same logic as Structured Text *)
(* Network 1 *)
CHARGING_SAFETY := CHARGER_IN AND NOT IGN_KEY;
(* Network 2 *)
IF SOC_BAT1 = 97 THEN BAT1_FULL := TRUE; END_IF;
IF SOC_BAT2 = 97 THEN BAT2_FULL := TRUE; END_IF;
IF SOC_BAT1 >= 80 THEN BAT1_80 := TRUE; END_IF;
IF SOC_BAT2 >= 80 THEN BAT2_80 := TRUE; END_IF;
(* Network 3 *)
CHARGE_1 := BAT1_80 AND BAT2_80;
(* Network 4 *)
RELAY1_TIMER(IN := CHARGING_SAFETY AND (NOT BAT1_CAN_ERROR OR BAT2_CAN_ERROR) AND (NOT BAT1_80 OR CHARGE_1) AND NOT BAT1_FULL AND NOT RELAY_BAT2 AND NOT ERROR_TIMER.Q, PT := T#2S);
RELAY_BAT1 := RELAY1_TIMER.Q OR CHARGER_IN AND BAT1_IGNITION AND NOT RELAY_BAT2 AND NOT BAT2_IGNITION;
(* Network 5 *)
RELAY2_TIMER(IN := CHARGING_SAFETY AND (NOT BAT2_CAN_ERROR OR BAT1_CAN_ERROR) AND (NOT BAT2_80 OR BAT1_FULL) AND NOT BAT2_FULL AND NOT RELAY_BAT1 AND NOT ERROR_TIMER.Q, PT := T#2S);
RELAY_BAT2 := RELAY2_TIMER.Q OR CHARGER_IN AND BAT2_IGNITION AND NOT RELAY_BAT1 AND NOT BAT1_IGNITION;
(* Network 6: Critical error -> turning of the ignition of the battery which is not charging -> indirectly turning on the ignition of both batteries *)
ERROR := BAT1_IGNITION AND RELAY_BAT2 OR BAT2_IGNITION AND RELAY_BAT1;
(* Network 7 *)
ERROR_TIMER(IN := ERROR, PT := T#2S);
END_FUNCTION_BLOCK

(* POU PROGRAM_FBs/DUAL_CLN_CHARGING, LD *)
FUNCTION_BLOCK DUAL_CLN_CHARGING
(*
THIS BLOCK IS COMPATIBLE FOR 2X CLN BATTERIES

Created BY: Adiga
Date: 8-08-24
Version: 1
 
*)

VAR_INPUT
	CHANNEL: BYTE;
	CHARGER_IN: BOOL;
	BAT_CAN_ERROR1: BOOL;
	BAT_CAN_ERROR2: BOOL;
	BAT1_IGN: BOOL;
	BAT2_IGN: BOOL;
	BATTERY_CHARGING: BOOL;

END_VAR

VAR_OUTPUT
	RELAY_BAT1: BOOL;
	RELAY_BAT2: BOOL;
	BLUE_LED_OUT: BOOL;
	ERROR: BOOL;
	BUZZER_ON: BOOL;
	CHARGING1: BOOL;
	CHARGING2: BOOL;
END_VAR

VAR
	CHARGE_1: BOOL;
	BAT_1_FULL: BOOL;
	BAT_2_FULL: BOOL;
	RX_SOLTERRA: RX_CAN;
	CHARGER_TIMER: TON;
	SOLTERRA_TX: CAN_TX;
	CHARGING_FRAME: ARRAY [0..7] OF BYTE  := 16#03,16#25,16#01,16#5E,0,0,0,0;

	T1: TON;
	T2: TON;
	T3: TON;
	SOC2: BYTE;
	SOC1: BYTE;
	TX_CLN: CAN_TX;
	IGNITION_OFF: BOOL;
	BAT_1_80: BOOL;
	BAT_2_80: BOOL;
	FTRIG1: F_TRIG;
	TIMER5: TON;
	T4: TON;
	T5: TON;

	CHARGE: F_TRIG;
END_VAR
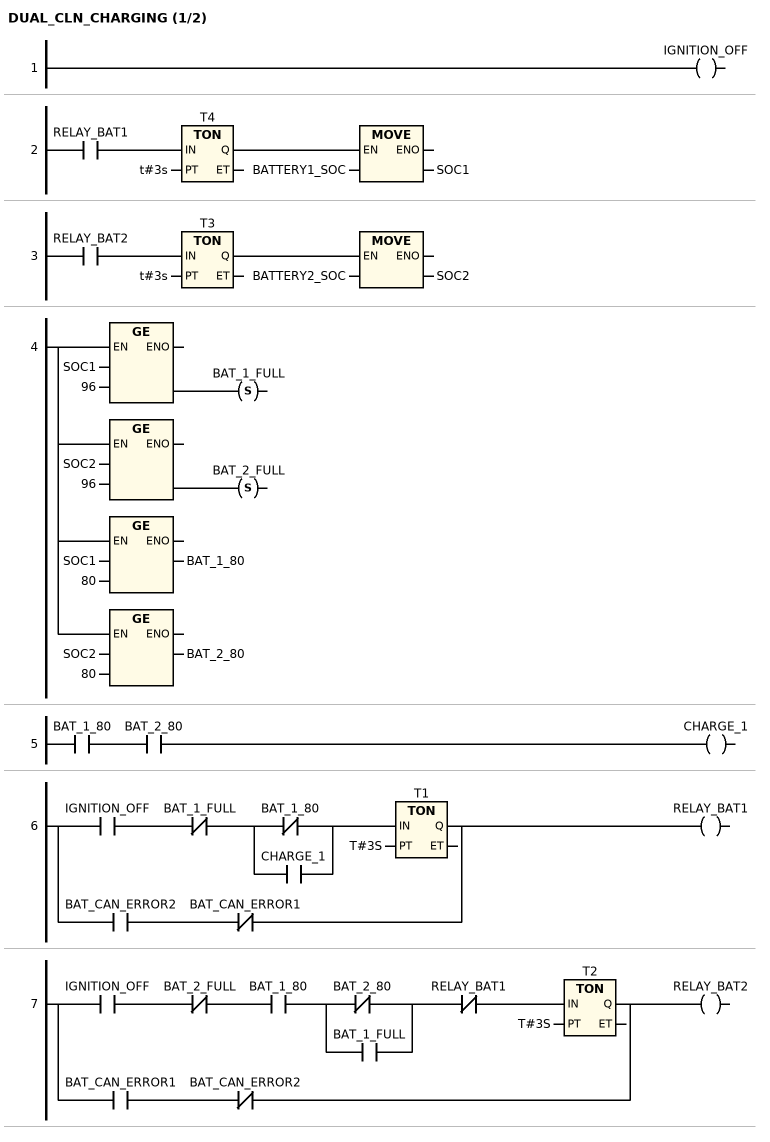
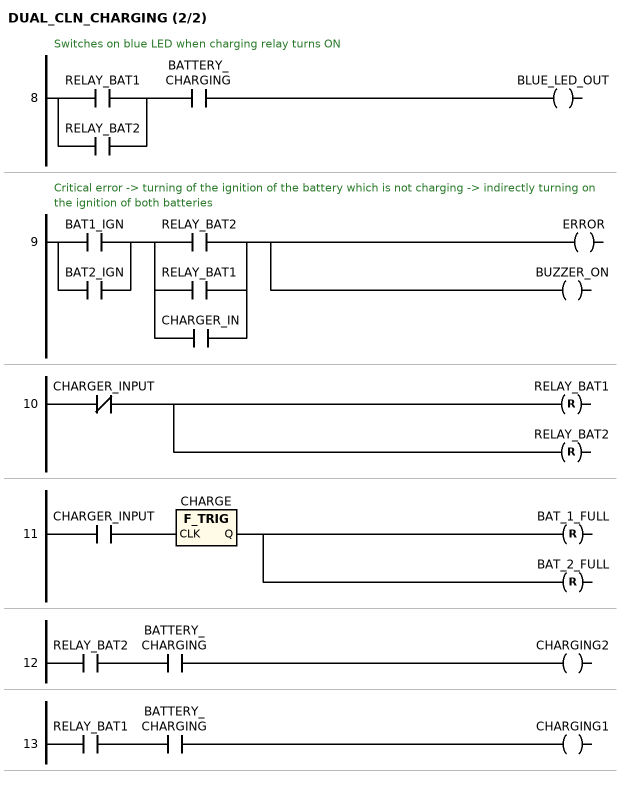
_LD_ (* Ladder Diagram *)
NETWORK 1
	* --- (IGNITION_OFF)
NETWORK 2
	[RELAY_BAT1] - T4:TON(IN: *, PT: t#3s)
		EN --- MOVE(BATTERY1_SOC) => SOC1
NETWORK 3
	[RELAY_BAT2] - T3:TON(IN: *, PT: t#3s)
		EN --- MOVE(BATTERY2_SOC) => SOC2
NETWORK 4
	*
		EN --- GE(SOC1, 96) => S BAT_1_FULL
		EN --- GE(SOC2, 96) => S BAT_2_FULL
		EN --- GE(SOC1, 80) => BAT_1_80
		EN --- GE(SOC2, 80) => BAT_2_80
NETWORK 5
	[BAT_1_80] - [BAT_2_80] --- (CHARGE_1)
NETWORK 6
	{ [IGNITION_OFF] - [/BAT_1_FULL] - { [/BAT_1_80] | [CHARGE_1] } - T1:TON(IN: *, PT: T#3S) | [BAT_CAN_ERROR2] - [/BAT_CAN_ERROR1] } --- (RELAY_BAT1)
NETWORK 7
	{ [IGNITION_OFF] - [/BAT_2_FULL] - [BAT_1_80] - { [/BAT_2_80] | [BAT_1_FULL] } - [/RELAY_BAT1] - T2:TON(IN: *, PT: T#3S) | [BAT_CAN_ERROR1] - [/BAT_CAN_ERROR2] } --- (RELAY_BAT2)
NETWORK 8 (* Switches on blue LED when charging relay turns ON *)
	{ [RELAY_BAT1] | [RELAY_BAT2] } - [BATTERY_CHARGING] --- (BLUE_LED_OUT)
NETWORK 9 (* Critical error -> turning of the ignition of the battery which is not charging -> indirectly turning on the ignition of both batteries *)
	{ [BAT1_IGN] | [BAT2_IGN] } - { [RELAY_BAT2] | [RELAY_BAT1] | [CHARGER_IN] } --- (ERROR) (BUZZER_ON)
NETWORK 10
	[/CHARGER_INPUT] --- (R RELAY_BAT1) (R RELAY_BAT2)
NETWORK 11
	[CHARGER_INPUT] - CHARGE:F_TRIG(CLK: *) --- (R BAT_1_FULL) (R BAT_2_FULL)
NETWORK 12
	[RELAY_BAT2] - [BATTERY_CHARGING] --- (CHARGING2)
NETWORK 13
	[RELAY_BAT1] - [BATTERY_CHARGING] --- (CHARGING1)
_END_LD_
(* the same logic as Structured Text *)
(* Network 1 *)
IGNITION_OFF := TRUE;
(* Network 2 *)
T4(IN := RELAY_BAT1, PT := t#3s);
IF T4.Q THEN
	SOC1 := BATTERY1_SOC;
END_IF;
(* Network 3 *)
T3(IN := RELAY_BAT2, PT := t#3s);
IF T3.Q THEN
	SOC2 := BATTERY2_SOC;
END_IF;
(* Network 4 *)
IF SOC1 >= 96 THEN BAT_1_FULL := TRUE; END_IF;
IF SOC2 >= 96 THEN BAT_2_FULL := TRUE; END_IF;
BAT_1_80 := SOC1 >= 80;
BAT_2_80 := SOC2 >= 80;
(* Network 5 *)
CHARGE_1 := BAT_1_80 AND BAT_2_80;
(* Network 6 *)
T1(IN := IGNITION_OFF AND NOT BAT_1_FULL AND (NOT BAT_1_80 OR CHARGE_1), PT := T#3S);
RELAY_BAT1 := T1.Q OR BAT_CAN_ERROR2 AND NOT BAT_CAN_ERROR1;
(* Network 7 *)
T2(IN := IGNITION_OFF AND NOT BAT_2_FULL AND BAT_1_80 AND (NOT BAT_2_80 OR BAT_1_FULL) AND NOT RELAY_BAT1, PT := T#3S);
RELAY_BAT2 := T2.Q OR BAT_CAN_ERROR1 AND NOT BAT_CAN_ERROR2;
(* Network 8: Switches on blue LED when charging relay turns ON *)
BLUE_LED_OUT := (RELAY_BAT1 OR RELAY_BAT2) AND BATTERY_CHARGING;
(* Network 9: Critical error -> turning of the ignition of the battery which is not charging -> indirectly turning on the ignition of both batteries *)
ERROR := (BAT1_IGN OR BAT2_IGN) AND (RELAY_BAT2 OR RELAY_BAT1 OR CHARGER_IN);
BUZZER_ON := ERROR;
(* Network 10 *)
IF NOT CHARGER_INPUT THEN RELAY_BAT1 := FALSE; RELAY_BAT2 := FALSE; END_IF;
(* Network 11 *)
CHARGE(CLK := CHARGER_INPUT);
IF CHARGE.Q THEN BAT_1_FULL := FALSE; BAT_2_FULL := FALSE; END_IF;
(* Network 12 *)
CHARGING2 := RELAY_BAT2 AND BATTERY_CHARGING;
(* Network 13 *)
CHARGING1 := RELAY_BAT1 AND BATTERY_CHARGING;
END_FUNCTION_BLOCK

(* POU EXCLUDES/IMU_SENSOR_HOLD, LD *)
FUNCTION_BLOCK IMU_SENSOR_HOLD
VAR_OUTPUT
	IMY_X_OUT: BYTE;
	IMU_Y_OUT: BYTE;
	IMU_BUZZER_ALERT: BOOL;
END_VAR
VAR
	RX_18C: RX_CAN;
	X_ANGLE_WORD: WORD;
	X_ANGLE: INT;
	Y_ANGLE_WORD: WORD;
	Y_ANGLE: INT;
	Y_IMU: INT;
	X_IMU: INT;
	TON_IMU: TON;
	Y_ALERT: BOOL;
	X_ALERT: BOOL;
	PAST_TIMER: TON;
	Y_PAST: INT;
	STORE_Y_MAX: BOOL;
	X_PAST: INT;
	STORE_X_MAX: BOOL;
	STORE_Y_MIN: BOOL;
	STORE_X_MIN: BOOL;
END_VAR
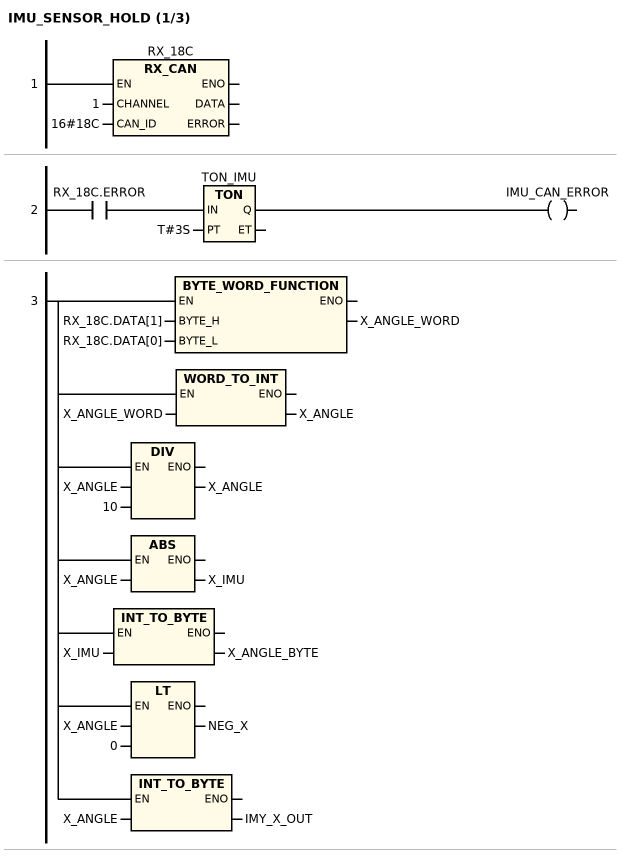
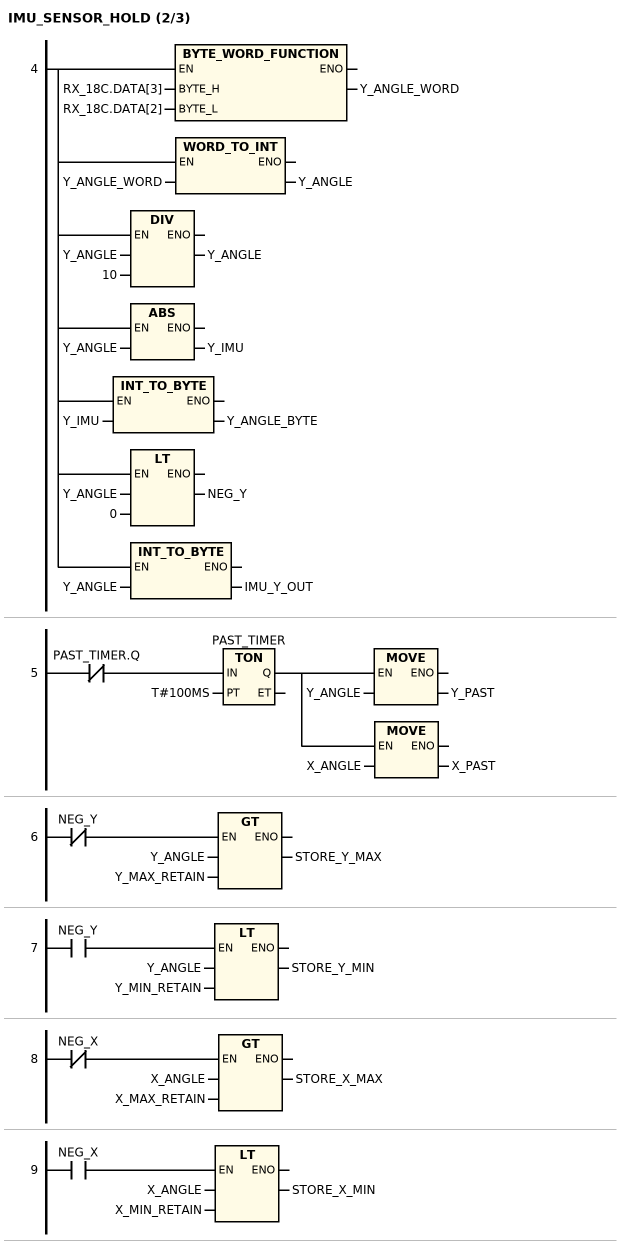
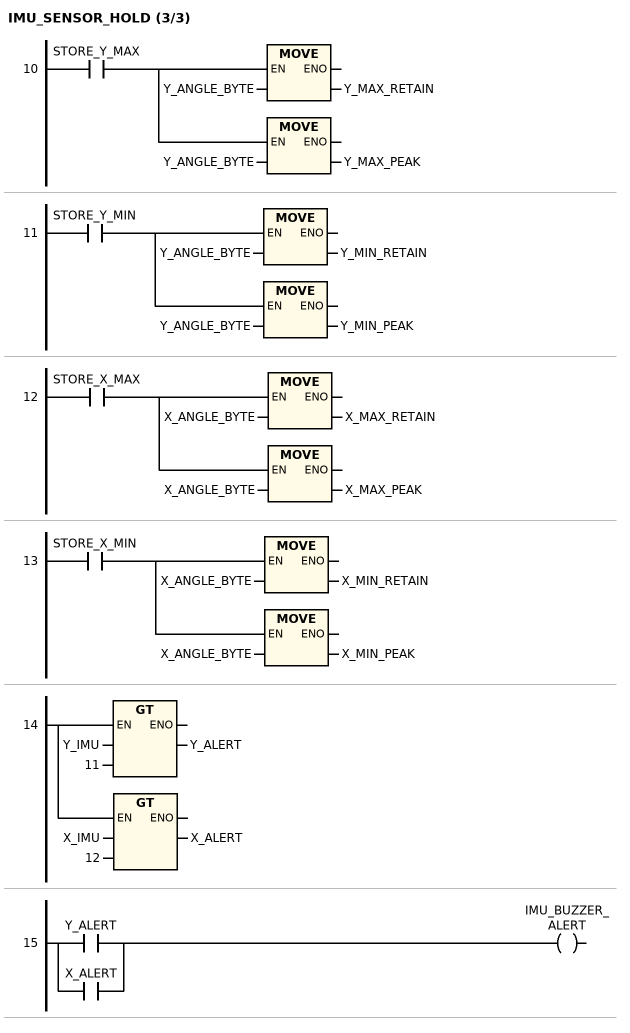
_LD_ (* Ladder Diagram *)
NETWORK 1
	*
		EN --- RX_18C:RX_CAN(CHANNEL: 1, CAN_ID: 16#18C)
NETWORK 2
	[RX_18C.ERROR] - TON_IMU:TON(IN: *, PT: T#3S) --- (IMU_CAN_ERROR)
NETWORK 3
	*
		EN --- BYTE_WORD_FUNCTION(BYTE_H: RX_18C.DATA[1], BYTE_L: RX_18C.DATA[0]) => X_ANGLE_WORD
		EN --- WORD_TO_INT(X_ANGLE_WORD) => X_ANGLE
		EN --- DIV(X_ANGLE, 10) => X_ANGLE
		EN --- ABS(X_ANGLE) => X_IMU
		EN --- INT_TO_BYTE(X_IMU) => X_ANGLE_BYTE
		EN --- LT(X_ANGLE, 0) => NEG_X
		EN --- INT_TO_BYTE(X_ANGLE) => IMY_X_OUT
NETWORK 4
	*
		EN --- BYTE_WORD_FUNCTION(BYTE_H: RX_18C.DATA[3], BYTE_L: RX_18C.DATA[2]) => Y_ANGLE_WORD
		EN --- WORD_TO_INT(Y_ANGLE_WORD) => Y_ANGLE
		EN --- DIV(Y_ANGLE, 10) => Y_ANGLE
		EN --- ABS(Y_ANGLE) => Y_IMU
		EN --- INT_TO_BYTE(Y_IMU) => Y_ANGLE_BYTE
		EN --- LT(Y_ANGLE, 0) => NEG_Y
		EN --- INT_TO_BYTE(Y_ANGLE) => IMU_Y_OUT
NETWORK 5
	[/PAST_TIMER.Q] - PAST_TIMER:TON(IN: *, PT: T#100MS)
		EN --- MOVE(Y_ANGLE) => Y_PAST
		EN --- MOVE(X_ANGLE) => X_PAST
NETWORK 6
	[/NEG_Y]
		EN --- GT(Y_ANGLE, Y_MAX_RETAIN) => STORE_Y_MAX
NETWORK 7
	[NEG_Y]
		EN --- LT(Y_ANGLE, Y_MIN_RETAIN) => STORE_Y_MIN
NETWORK 8
	[/NEG_X]
		EN --- GT(X_ANGLE, X_MAX_RETAIN) => STORE_X_MAX
NETWORK 9
	[NEG_X]
		EN --- LT(X_ANGLE, X_MIN_RETAIN) => STORE_X_MIN
NETWORK 10
	[STORE_Y_MAX]
		EN --- MOVE(Y_ANGLE_BYTE) => Y_MAX_RETAIN
		EN --- MOVE(Y_ANGLE_BYTE) => Y_MAX_PEAK
NETWORK 11
	[STORE_Y_MIN]
		EN --- MOVE(Y_ANGLE_BYTE) => Y_MIN_RETAIN
		EN --- MOVE(Y_ANGLE_BYTE) => Y_MIN_PEAK
NETWORK 12
	[STORE_X_MAX]
		EN --- MOVE(X_ANGLE_BYTE) => X_MAX_RETAIN
		EN --- MOVE(X_ANGLE_BYTE) => X_MAX_PEAK
NETWORK 13
	[STORE_X_MIN]
		EN --- MOVE(X_ANGLE_BYTE) => X_MIN_RETAIN
		EN --- MOVE(X_ANGLE_BYTE) => X_MIN_PEAK
NETWORK 14
	*
		EN --- GT(Y_IMU, 11) => Y_ALERT
		EN --- GT(X_IMU, 12) => X_ALERT
NETWORK 15
	{ [Y_ALERT] | [X_ALERT] } --- (IMU_BUZZER_ALERT)
_END_LD_
(* the same logic as Structured Text *)
(* Network 1 *)
RX_18C(CHANNEL := 1, CAN_ID := 16#18C);
(* Network 2 *)
TON_IMU(IN := RX_18C.ERROR, PT := T#3S);
IMU_CAN_ERROR := TON_IMU.Q;
(* Network 3 *)
X_ANGLE_WORD := BYTE_WORD_FUNCTION(BYTE_H := RX_18C.DATA[1], BYTE_L := RX_18C.DATA[0]);
X_ANGLE := WORD_TO_INT(X_ANGLE_WORD);
X_ANGLE := X_ANGLE / 10;
X_IMU := ABS(X_ANGLE);
X_ANGLE_BYTE := INT_TO_BYTE(X_IMU);
NEG_X := X_ANGLE < 0;
IMY_X_OUT := INT_TO_BYTE(X_ANGLE);
(* Network 4 *)
Y_ANGLE_WORD := BYTE_WORD_FUNCTION(BYTE_H := RX_18C.DATA[3], BYTE_L := RX_18C.DATA[2]);
Y_ANGLE := WORD_TO_INT(Y_ANGLE_WORD);
Y_ANGLE := Y_ANGLE / 10;
Y_IMU := ABS(Y_ANGLE);
Y_ANGLE_BYTE := INT_TO_BYTE(Y_IMU);
NEG_Y := Y_ANGLE < 0;
IMU_Y_OUT := INT_TO_BYTE(Y_ANGLE);
(* Network 5 *)
PAST_TIMER(IN := NOT PAST_TIMER.Q, PT := T#100MS);
IF PAST_TIMER.Q THEN
	Y_PAST := Y_ANGLE;
	X_PAST := X_ANGLE;
END_IF;
(* Network 6 *)
IF NOT NEG_Y THEN
	STORE_Y_MAX := Y_ANGLE > Y_MAX_RETAIN;
END_IF;
(* Network 7 *)
IF NEG_Y THEN
	STORE_Y_MIN := Y_ANGLE < Y_MIN_RETAIN;
END_IF;
(* Network 8 *)
IF NOT NEG_X THEN
	STORE_X_MAX := X_ANGLE > X_MAX_RETAIN;
END_IF;
(* Network 9 *)
IF NEG_X THEN
	STORE_X_MIN := X_ANGLE < X_MIN_RETAIN;
END_IF;
(* Network 10 *)
IF STORE_Y_MAX THEN
	Y_MAX_RETAIN := Y_ANGLE_BYTE;
	Y_MAX_PEAK := Y_ANGLE_BYTE;
END_IF;
(* Network 11 *)
IF STORE_Y_MIN THEN
	Y_MIN_RETAIN := Y_ANGLE_BYTE;
	Y_MIN_PEAK := Y_ANGLE_BYTE;
END_IF;
(* Network 12 *)
IF STORE_X_MAX THEN
	X_MAX_RETAIN := X_ANGLE_BYTE;
	X_MAX_PEAK := X_ANGLE_BYTE;
END_IF;
(* Network 13 *)
IF STORE_X_MIN THEN
	X_MIN_RETAIN := X_ANGLE_BYTE;
	X_MIN_PEAK := X_ANGLE_BYTE;
END_IF;
(* Network 14 *)
Y_ALERT := Y_IMU > 11;
X_ALERT := X_IMU > 12;
(* Network 15 *)
IMU_BUZZER_ALERT := Y_ALERT OR X_ALERT;
END_FUNCTION_BLOCK

(* POU FUNCTIONS/MAP_INT, ST *)
FUNCTION MAP_INT : INT
(*
Created By: Nikshitha S
Date: 10-08-2023
Version: 1
Description: This function block maps the Input value range to the Output value range for the values in INT datatype.
Thus, consuming less memory than the library block "LIN_TRAFO" which uses REAL datatype.
*)
VAR_INPUT
	IN: INT;
	IN_MIN:INT;
	IN_MAX : INT;
	OUT_MIN:INT;
	OUT_MAX:INT;
END_VAR
VAR
	ERROR: BOOL;
	FINAL_MAP: INT;
	INPUT_RANGE: INT;
	OUTPUT_RANGE: INT;
END_VAR
ERROR := (IN_MAX-IN_MIN=0) OR (IN<IN_MIN) OR (IN>IN_MAX);
INPUT_RANGE := IN_MAX-IN_MIN;
OUTPUT_RANGE := OUT_MAX-OUT_MIN;
MAP_INT:= ((IN-IN_MIN)*OUTPUT_RANGE) / INPUT_RANGE + OUT_MIN;
IF ERROR AND (IN<IN_MIN)THEN
MAP_INT:=OUT_MIN;
END_IF
IF ERROR AND (IN>IN_MAX)THEN
MAP_INT:=OUT_MAX;
END_IF
END_FUNCTION

(* POU EXCLUDES/MAP_REAL, ST *)
FUNCTION MAP_REAL : REAL
(*
Created By: Bhagyesh
Date: Nov - 2021
Description: This function block maps the Input value range to the Output value range for the values in REAL datatype.
*)
VAR_INPUT
	IN: REAL;				(* input value*)
	IN_MIN:REAL;			(* minimum input value *)
	IN_MAX:REAL;			(* maximum input value *)
	OUT_MIN:REAL;		(* corresponding minimum output value *)
	OUT_MAX:REAL;		(* corresponding maximum output value *)
END_VAR
VAR
	Diff: REAL;
	ERROR: BOOL;		(* error: IN_MIN = IN_MAX or IN out of interval *)
END_VAR
Diff := IN_MAX-IN_MIN;
ERROR := (Diff=0) OR (IN<IN_MIN) OR (IN>IN_MAX);
MAP_REAL:= (IN-IN_MIN)/Diff * (OUT_MAX-OUT_MIN) + OUT_MIN;
IF ERROR AND (IN<IN_MIN)THEN
MAP_REAL:=OUT_MIN;
END_IF
IF ERROR AND (IN>IN_MAX)THEN
MAP_REAL:=OUT_MAX;
END_IF
END_FUNCTION

(* Visualisation GLX_v3
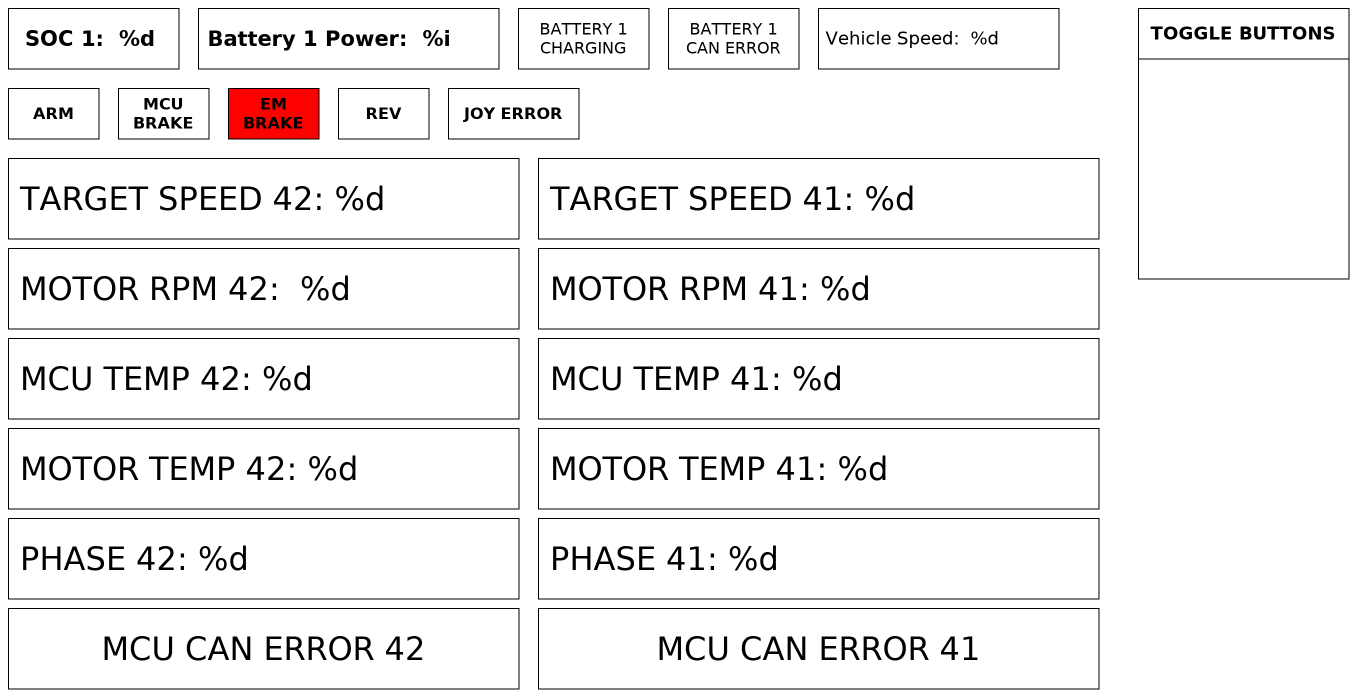
rounded rectangle at (10,10)-(181,71): text "SOC 1:  %d"; shows .BATTERY1_SOC
rounded rectangle at (200,10)-(501,71): text "Battery 1 Power:  %i"; shows .BATTERY1_POWER
rounded rectangle at (820,10)-(1061,71): text "Vehicle Speed:  %d"; shows .SPEED
rounded rectangle at (10,90)-(101,141): text "ARM"; alarm colour if .MCU_IGNITION
rounded rectangle at (120,90)-(211,141): text "MCU / BRAKE"; alarm colour if .MCU_BRAKE
rounded rectangle at (230,90)-(321,141): text "EM / BRAKE"; alarm colour if .EM_BRAKE
rounded rectangle at (540,250)-(1101,331): text "MOTOR RPM 41: %d"; shows .MOTOR_RPM[1]
rounded rectangle at (10,250)-(521,331): text "MOTOR RPM 42:  %d"; shows .MOTOR_RPM[2]
rounded rectangle at (540,340)-(1101,421): text "MCU TEMP 41: %d"; shows .MCU_TEMPERATURE[1]
rounded rectangle at (10,340)-(521,421): text "MCU TEMP 42: %d"; shows .MCU_TEMPERATURE[2]
rounded rectangle at (540,520)-(1101,601): text "PHASE 41: %d"; shows .MOTOR_PHASE_CURRENT[1]
rounded rectangle at (10,520)-(521,601): text "PHASE 42: %d"; shows .MOTOR_PHASE_CURRENT[2]
rounded rectangle at (540,160)-(1101,241): text "TARGET SPEED 41: %d"; shows .MOTOR_TARGET_RPM[1]
rounded rectangle at (10,160)-(521,241): text "TARGET SPEED 42: %d"; shows .MOTOR_TARGET_RPM[2]
rounded rectangle at (450,90)-(581,141): text "JOY ERROR"; alarm colour if .JOY_ERROR
rounded rectangle at (10,610)-(521,691): text "MCU CAN ERROR 42"; alarm colour if .MCU_CAN_ERROR[2]
rounded rectangle at (670,10)-(801,71): text "BATTERY 1 / CAN ERROR"; alarm colour if .BATTERY1_CAN_ERROR
rounded rectangle at (340,90)-(431,141): text "REV"; alarm colour if .REVERSE
rounded rectangle at (520,10)-(651,71): text "BATTERY 1 / CHARGING"; alarm colour if .BATTERY1_CHARGING
rounded rectangle at (540,610)-(1101,691): text "MCU CAN ERROR 41"; alarm colour if .MCU_CAN_ERROR[1]
rounded rectangle at (540,430)-(1101,511): text "MOTOR TEMP 41: %d"; shows .MOTOR_TEMPERATURE[1]
rounded rectangle at (10,430)-(521,511): text "MOTOR TEMP 42: %d"; shows .MOTOR_TEMPERATURE[2]
rectangle at (1140,10)-(1351,61): text "TOGGLE BUTTONS"
1 more shapes without text or variables
*)
